(* Publish stable source identities and the complete typed Sequence status. *)
stMotionIntent.udiZCommandId := udiZCommandId;
stMotionIntent.udiRCommandId := udiRCommandId;
GVL_Status.stFast.stSequence.nAcceptedCommandId := udiActiveStartCommandId;
GVL_Status.stFast.stSequence.bBusy := bBusy;
GVL_Status.stFast.stSequence.bDone := bDone;
GVL_Status.stFast.stSequence.bAborted := bAborted;
GVL_Status.stFast.stSequence.bError := bError;
GVL_Status.stFast.stSequence.nErrorId := udiFirstFaultId;
GVL_Status.stFast.stSequence.eState := eNextState;
GVL_Status.stFast.stSequence.eStep := eStep;
GVL_Status.stFast.stSequence.eSubPhase := eSubPhase;
GVL_Status.stFast.stSequence.eEndCause := eEndCause;
GVL_Status.stFast.stSequence.eExitIntent := eExitIntent;
GVL_Status.stFast.stSequence.bCycleNok := bCycleNokLatched;
GVL_Status.stFast.stSequence.bRpmStopped := bRpmStopped;
GVL_Status.stFast.stSequence.bForceInBand := bForceInBand;
GVL_Status.stFast.stSequence.rStepTime_s := rStepTime_s;
GVL_Status.stFast.stSequence.rQualifiedForceHoldTime_s := rQualifiedForceHoldTime_s;
GVL_Status.stFast.stSequence.rForceSet_kN := rForceSet_kN;
GVL_Status.stFast.stSequence.rForceRamp_kN_s := rForceRamp_kN_s;
GVL_Status.stFast.stSequence.bForceControlEnable := bForceControlEnable;
GVL_Status.stFast.stSequence.bForceProfileTransfer := bForceProfileTransfer;
GVL_Status.stFast.stSequence.rForceTransferVelocity_mm_s := rForceTransferVelocity_mm_s;
GVL_Status.stFast.stSequence.rTargetRelativePosition_mm := rTargetRelativePosition_mm;
GVL_Status.stFast.stSequence.rHardMaximumRelativePosition_mm := rHardMaximumRelativePosition_mm;
GVL_Status.stFast.stSequence.bForceHardLimitActive := bHardForceActive;
GVL_Status.stFast.stSequence.bStrokeHardLimitActive := bHardStrokeActive;
GVL_Status.stFast.stSequence.bCollisionLimitActive := bCollisionLimitActive;
GVL_Status.stFast.stSequence.rSpeedSet_rpm := rSpeedSet_rpm;
GVL_Status.stFast.stSequence.stContact := fbContactDetect.stOutput;
GVL_Status.stFast.stSequence.stForceDecline := fbForceDecline.stOutput;
GVL_Status.stFast.stSequence.stStepCriterion := fbStepCriterion.stOutput;
GVL_Status.stFast.stSequence.stMotionIntent := stMotionIntent;
GVL_Status.stFast.stSequence.stFastConfigSnapshot := stFastConfigSnapshot;

GVL_Alarm.astRequests[9].eCode := E_AlarmCode.ALARM_CFF_CRITERION_FAULT;
GVL_Alarm.astRequests[9].eLevel := E_AlarmLevel.ALARM_LEVEL_FAULT;
GVL_Alarm.astRequests[9].nTextId := 3000;
GVL_Alarm.astRequests[9].nSourceId := 9;
GVL_Alarm.astRequests[9].bLatch := TRUE;
GVL_Alarm.astRequests[9].bActive := fbContactDetect.stOutput.bFault
    OR fbForceDecline.stOutput.bFault
    OR fbStepCriterion.stOutput.bFault;
GVL_Alarm.astRequests[10].eCode := E_AlarmCode.ALARM_CFF_SEQUENCE_FAULT;
GVL_Alarm.astRequests[10].eLevel := E_AlarmLevel.ALARM_LEVEL_FAULT;
GVL_Alarm.astRequests[10].nTextId := 3200;
GVL_Alarm.astRequests[10].nSourceId := 10;
GVL_Alarm.astRequests[10].bLatch := TRUE;
GVL_Alarm.astRequests[10].bActive := udiFirstFaultId <> 0;

(* Exactly one state assignment completes the scan. *)
ePreviousState := eState;
eState := eNextState;
bStateEntry := eState <> ePreviousState;

END_PROGRAM

// ---- POUs/FunctionBlocks/Control/FB_ForceDeclineObserver.TcPOU
FUNCTION_BLOCK FB_ForceDeclineObserver
VAR_INPUT
    (* 调用者完整赋值的Force Decline输入。 *)
    stInput : ST_ForceDeclineInput;
END_VAR
VAR_OUTPUT
    (* Arm、候选、确认、导数、锁存和故障输出。 *)
    stOutput : ST_ForceDeclineOutput;
END_VAR
VAR
    (* 当前步骤已经达到Arm Force。 *)
    bArmed : BOOL;
    (* 当前保持Decline回差候选。 *)
    bCandidate : BOOL;
    (* Decline已经连续确认。 *)
    bConfirmed : BOOL;
    (* 已获得上一个有效力样本。 *)
    bPreviousSampleValid : BOOL;
    (* 当前扫描满足全部Decline确认条件。 *)
    bDeclineCondition : BOOL;
    (* 当前配置和输入均有效。 *)
    bConfigurationValid : BOOL;
    (* 算法故障锁存；只有显式Reset清除。 *)
    bFaultLatched : BOOL;
    (* 已锁存的确定性故障编号。 *)
    udiLatchedFaultId : UDINT;
    (* 上一个有效力样本，单位kN。 *)
    rPreviousForce_kN : LREAL;
    (* 相邻样本力变化率，单位kN/s。 *)
    rForceDerivative_kN_s : LREAL;
    (* 连续确认累计时间，单位s。 *)
    rStableTime_s : LREAL;
    (* 确认锁存力，单位kN。 *)
    rLatchedForce_kN : LREAL;
    (* 确认锁存累计S_rel，单位mm。 *)
    rLatchedRelativePosition_mm : LREAL;
    (* 确认锁存主轴转速，单位rpm。 *)
    rLatchedSpeed_rpm : LREAL;
    (* 确认锁存步骤时间，单位s。 *)
    rLatchedStepTime_s : LREAL;
END_VAR

(* ---------------------------------------------------------
   Force Decline观察器。
   进入：步骤选择Decline主判据并提供有效ForceCriterion、RPM、S_rel和速度。
   动作：先Arm，再要求负下降率、窗口、捕获速度和连续Debounce。
   成功：锁存确认事实；不关闭PI、不切换Profile、不写流程状态。
   Fault：配置、信号或数值无效时锁存，只有显式Reset清除。
   --------------------------------------------------------- *)
IF stInput.bReset THEN
    bArmed := FALSE;
    bCandidate := FALSE;
    bConfirmed := FALSE;
    bPreviousSampleValid := FALSE;
    bFaultLatched := FALSE;
    udiLatchedFaultId := 0;
    rPreviousForce_kN := 0.0;
    rForceDerivative_kN_s := 0.0;
    rStableTime_s := 0.0;
    rLatchedForce_kN := 0.0;
    rLatchedRelativePosition_mm := 0.0;
    rLatchedSpeed_rpm := 0.0;
    rLatchedStepTime_s := 0.0;
ELSIF NOT stInput.bEnable THEN
    (* Disable结束当前步骤观察窗口，但故障保持到Reset。 *)
    bArmed := FALSE;
    bCandidate := FALSE;
    bConfirmed := FALSE;
    bPreviousSampleValid := FALSE;
    rForceDerivative_kN_s := 0.0;
    rStableTime_s := 0.0;
ELSIF NOT bFaultLatched AND NOT bConfirmed THEN
    bConfigurationValid := stInput.bSignalValid
        AND FC_IsFiniteLReal(rValue := stInput.rForceActual_kN)
        AND FC_IsFiniteLReal(rValue := stInput.rSpeed_rpm)
        AND FC_IsFiniteLReal(rValue := stInput.rRelativePosition_mm)
        AND FC_IsFiniteLReal(rValue := stInput.rAxisVelocity_mm_s)
        AND FC_IsFiniteLReal(rValue := stInput.rStepTime_s)
        AND FC_IsFiniteLReal(rValue := stInput.rArmForce_kN)
        AND FC_IsFiniteLReal(rValue := stInput.rDeclineTo_kN)
        AND FC_IsFiniteLReal(rValue := stInput.rHysteresis_kN)
        AND FC_IsFiniteLReal(rValue := stInput.rMinimumDeclineRate_kN_s)
        AND FC_IsFiniteLReal(rValue := stInput.rCriterionSRelMinimum_mm)
        AND FC_IsFiniteLReal(rValue := stInput.rCriterionSRelMaximum_mm)
        AND FC_IsFiniteLReal(rValue := stInput.rCriterionRpmMinimum)
        AND FC_IsFiniteLReal(rValue := stInput.rCaptureMaximumVelocity_mm_s)
        AND FC_IsFiniteLReal(rValue := stInput.rDebounceTime_s)
        AND FC_IsFiniteLReal(rValue := stInput.rCycleTime_s)
        AND (stInput.rDeclineTo_kN >= 0.0)
        AND (stInput.rHysteresis_kN >= 0.0)
        AND (stInput.rArmForce_kN > stInput.rDeclineTo_kN + stInput.rHysteresis_kN)
        AND (stInput.rMinimumDeclineRate_kN_s > 0.0)
        AND (stInput.rCriterionSRelMaximum_mm >= stInput.rCriterionSRelMinimum_mm)
        AND (stInput.rCriterionRpmMinimum >= 0.0)
        AND (stInput.rCaptureMaximumVelocity_mm_s > 0.0)
        AND (stInput.rDebounceTime_s > 0.0)
        AND (stInput.rCycleTime_s > 0.0);

    IF NOT bConfigurationValid THEN
        bFaultLatched := TRUE;
        udiLatchedFaultId := 16#00009101;
    ELSE
        IF bPreviousSampleValid THEN
            rForceDerivative_kN_s := (stInput.rForceActual_kN - rPreviousForce_kN)
                / stInput.rCycleTime_s;
            IF NOT FC_IsFiniteLReal(rValue := rForceDerivative_kN_s) THEN
                bFaultLatched := TRUE;
                udiLatchedFaultId := 16#00009102;
            END_IF
        ELSE
            rForceDerivative_kN_s := 0.0;
            bPreviousSampleValid := TRUE;
        END_IF
        rPreviousForce_kN := stInput.rForceActual_kN;

        IF NOT bFaultLatched THEN
            IF stInput.rForceActual_kN >= stInput.rArmForce_kN THEN
                bArmed := TRUE;
            END_IF

            IF NOT bCandidate AND bArmed
                AND (stInput.rForceActual_kN <= stInput.rDeclineTo_kN) THEN
                bCandidate := TRUE;
            END_IF

            IF bCandidate AND (stInput.rForceActual_kN
                > stInput.rDeclineTo_kN + stInput.rHysteresis_kN) THEN
                bCandidate := FALSE;
                rStableTime_s := 0.0;
            ELSE
                bDeclineCondition := bCandidate
                    AND (stInput.rForceActual_kN <= stInput.rDeclineTo_kN)
                    AND (rForceDerivative_kN_s <= -ABS(stInput.rMinimumDeclineRate_kN_s))
                    AND (stInput.rRelativePosition_mm >= stInput.rCriterionSRelMinimum_mm)
                    AND (stInput.rRelativePosition_mm <= stInput.rCriterionSRelMaximum_mm)
                    AND (ABS(stInput.rSpeed_rpm) >= ABS(stInput.rCriterionRpmMinimum))
                    AND (ABS(stInput.rAxisVelocity_mm_s) <= ABS(stInput.rCaptureMaximumVelocity_mm_s));

                IF bDeclineCondition THEN
                    rStableTime_s := rStableTime_s + stInput.rCycleTime_s;
                    IF NOT FC_IsFiniteLReal(rValue := rStableTime_s) THEN
                        bFaultLatched := TRUE;
                        udiLatchedFaultId := 16#00009103;
                    ELSIF rStableTime_s >= stInput.rDebounceTime_s THEN
                        bCandidate := FALSE;
                        bConfirmed := TRUE;
                        rLatchedForce_kN := stInput.rForceActual_kN;
                        rLatchedRelativePosition_mm := stInput.rRelativePosition_mm;
                        rLatchedSpeed_rpm := stInput.rSpeed_rpm;
                        rLatchedStepTime_s := stInput.rStepTime_s;
                    END_IF
                ELSE
                    (* 任一连续确认条件中断均清零Debounce；候选只由Force回差释放。 *)
                    rStableTime_s := 0.0;
                END_IF
            END_IF
        END_IF
    END_IF
END_IF

stOutput.bArmed := bArmed;
stOutput.bCandidate := bCandidate;
stOutput.bConfirmed := bConfirmed;
stOutput.rForceDerivative_kN_s := rForceDerivative_kN_s;
stOutput.rStableTime_s := rStableTime_s;
stOutput.rLatchedForce_kN := rLatchedForce_kN;
stOutput.rLatchedRelativePosition_mm := rLatchedRelativePosition_mm;
stOutput.rLatchedSpeed_rpm := rLatchedSpeed_rpm;
stOutput.rLatchedStepTime_s := rLatchedStepTime_s;
stOutput.bFault := bFaultLatched;
stOutput.nFaultId := udiLatchedFaultId;

END_FUNCTION_BLOCK

// ---- POUs/FunctionBlocks/Control/FB_StepProceedingCriterion.TcPOU
FUNCTION_BLOCK FB_StepProceedingCriterion
VAR_INPUT
    (* 调用者完整赋值的步骤推进输入。 *)
    stInput : ST_StepCriterionInput;
END_VAR
VAR_OUTPUT
    (* 步骤结束事实、动作、锁存和故障输出。 *)
    stOutput : ST_StepCriterionOutput;
END_VAR
VAR
    (* 当前Primary已经满足。 *)
    bPrimaryMet : BOOL;
    (* 当前Primary需要累计S_rel Secondary。 *)
    bSecondaryRequired : BOOL;
    (* 本扫描输入数值和配置有效。 *)
    bConfigurationValid : BOOL;
    (* 算法故障锁存；只有显式Reset清除。 *)
    bFaultLatched : BOOL;
    (* 已锁存的确定性故障编号。 *)
    udiLatchedFaultId : UDINT;
END_VAR

(* ---------------------------------------------------------
   步骤推进判据。
   进入：单一Primary、可选累计S_rel Secondary、StepMin/Max和硬原因有效。
   动作：安全原因和Secondary优先，Primary满足立即结束，StepMax只监视未满足Primary。
   成功：锁存EndCause、Force、S_rel、时间和流程动作。
   Fault：配置、数值或未知枚举无效时锁存，只有显式Reset清除。
   --------------------------------------------------------- *)
IF stInput.bReset THEN
    stOutput.bArmed := FALSE;
    stOutput.bPrimaryMet := FALSE;
    stOutput.bSecondaryLimitReached := FALSE;
    stOutput.bEndConfirmed := FALSE;
    stOutput.bTooShort := FALSE;
    stOutput.bNok := FALSE;
    stOutput.bAdvanceRequested := FALSE;
    stOutput.bControlledExitRequested := FALSE;
    stOutput.bDownwardMotionInhibited := FALSE;
    stOutput.eEndCause := STEP_END_NONE;
    stOutput.rLatchedForce_kN := 0.0;
    stOutput.rLatchedRelativePosition_mm := 0.0;
    stOutput.rLatchedStepTime_s := 0.0;
    stOutput.bFault := FALSE;
    stOutput.nFaultId := 0;
    bFaultLatched := FALSE;
    udiLatchedFaultId := 0;
    RETURN;
END_IF

IF NOT stInput.bEnable THEN
    stOutput.bArmed := FALSE;
    RETURN;
END_IF

stOutput.bArmed := stInput.bForceDeclineArmed;
IF bFaultLatched THEN
    stOutput.bEndConfirmed := TRUE;
    stOutput.bNok := TRUE;
    stOutput.bAdvanceRequested := FALSE;
    stOutput.bControlledExitRequested := TRUE;
    stOutput.bDownwardMotionInhibited := TRUE;
    stOutput.eEndCause := STEP_END_NONE;
    stOutput.bFault := TRUE;
    stOutput.nFaultId := udiLatchedFaultId;
    RETURN;
END_IF
IF stOutput.bEndConfirmed THEN
    RETURN;
END_IF

bConfigurationValid := FC_IsFiniteLReal(rValue := stInput.rRelativePosition_mm)
    AND FC_IsFiniteLReal(rValue := stInput.rRelativeDistanceTarget_mm)
    AND FC_IsFiniteLReal(rValue := stInput.rStepTime_s)
    AND FC_IsFiniteLReal(rValue := stInput.rStepTimeTarget_s)
    AND FC_IsFiniteLReal(rValue := stInput.rStepMinimumTime_s)
    AND FC_IsFiniteLReal(rValue := stInput.rStepMaximumTime_s)
    AND FC_IsFiniteLReal(rValue := stInput.rForceActual_kN)
    AND FC_IsFiniteLReal(rValue := stInput.rSecondaryDistanceLimit_mm)
    AND (stInput.rStepTime_s >= 0.0)
    AND (stInput.rStepMinimumTime_s >= 0.0)
    AND (stInput.rStepMaximumTime_s > 0.0)
    AND (stInput.rStepMinimumTime_s <= stInput.rStepMaximumTime_s)
    AND NOT (stInput.bForceDeclineConfirmed AND NOT stInput.bForceDeclineArmed);
IF NOT bConfigurationValid THEN
    bFaultLatched := TRUE;
    udiLatchedFaultId := 16#00009201;
END_IF
IF bFaultLatched THEN
    stOutput.bEndConfirmed := TRUE;
    stOutput.bNok := TRUE;
    stOutput.bAdvanceRequested := FALSE;
    stOutput.bControlledExitRequested := TRUE;
    stOutput.bDownwardMotionInhibited := TRUE;
    stOutput.eEndCause := STEP_END_NONE;
    stOutput.bFault := TRUE;
    stOutput.nFaultId := udiLatchedFaultId;
    RETURN;
END_IF

CASE stInput.ePrimaryCriterion OF
    STEP_CRIT_RELATIVE_DISTANCE:
        bSecondaryRequired := FALSE;
        bPrimaryMet := stInput.rRelativePosition_mm >= stInput.rRelativeDistanceTarget_mm;
        IF stInput.rRelativeDistanceTarget_mm <= 0.0 THEN
            bFaultLatched := TRUE;
            udiLatchedFaultId := 16#00009202;
        END_IF
    STEP_CRIT_STEP_TIME:
        bSecondaryRequired := TRUE;
        bPrimaryMet := stInput.rStepTime_s >= stInput.rStepTimeTarget_s;
        IF (stInput.rStepTimeTarget_s <= 0.0)
            OR (stInput.rStepTimeTarget_s < stInput.rStepMinimumTime_s)
            OR (stInput.rStepTimeTarget_s > stInput.rStepMaximumTime_s)
            OR (stInput.rSecondaryDistanceLimit_mm <= 0.0) THEN
            bFaultLatched := TRUE;
            udiLatchedFaultId := 16#00009203;
        END_IF
    STEP_CRIT_FORCE_DECLINE_TO:
        bSecondaryRequired := TRUE;
        bPrimaryMet := stInput.bForceDeclineConfirmed;
        IF stInput.rSecondaryDistanceLimit_mm <= 0.0 THEN
            bFaultLatched := TRUE;
            udiLatchedFaultId := 16#00009204;
        END_IF
ELSE
    bFaultLatched := TRUE;
    udiLatchedFaultId := 16#00009205;
END_CASE

IF NOT bFaultLatched AND bSecondaryRequired THEN
    CASE stInput.eSecondaryAction OF
        SECONDARY_ADVANCE_AND_NOK:
        SECONDARY_CONTROLLED_EXIT_NOK:
    ELSE
        bFaultLatched := TRUE;
        udiLatchedFaultId := 16#00009206;
    END_CASE
END_IF
IF bFaultLatched THEN
    stOutput.bEndConfirmed := TRUE;
    stOutput.bNok := TRUE;
    stOutput.bAdvanceRequested := FALSE;
    stOutput.bControlledExitRequested := TRUE;
    stOutput.bDownwardMotionInhibited := TRUE;
    stOutput.eEndCause := STEP_END_NONE;
    stOutput.bFault := TRUE;
    stOutput.nFaultId := udiLatchedFaultId;
    RETURN;
END_IF

(* EVAL_STAGE_HARD_CAUSE：Stop、轴、传感器和硬边界拥有最高优先级。 *)
IF stInput.bStopRequested THEN
    stOutput.bEndConfirmed := TRUE;
    stOutput.bNok := TRUE;
    stOutput.bControlledExitRequested := TRUE;
    stOutput.bDownwardMotionInhibited := TRUE;
    stOutput.eEndCause := STEP_END_STOP_REQUEST;
ELSIF stInput.bAxisFault THEN
    stOutput.bEndConfirmed := TRUE;
    stOutput.bNok := TRUE;
    stOutput.bControlledExitRequested := TRUE;
    stOutput.bDownwardMotionInhibited := TRUE;
    stOutput.eEndCause := STEP_END_AXIS_FAULT;
ELSIF stInput.bSensorInvalid OR NOT stInput.bSignalValid THEN
    stOutput.bEndConfirmed := TRUE;
    stOutput.bNok := TRUE;
    stOutput.bControlledExitRequested := TRUE;
    stOutput.bDownwardMotionInhibited := TRUE;
    stOutput.eEndCause := STEP_END_SENSOR_INVALID;
ELSIF stInput.bCollisionActive THEN
    stOutput.bEndConfirmed := TRUE;
    stOutput.bNok := TRUE;
    stOutput.bControlledExitRequested := TRUE;
    stOutput.bDownwardMotionInhibited := TRUE;
    stOutput.eEndCause := STEP_END_COLLISION;
ELSIF stInput.bHardForceActive THEN
    stOutput.bEndConfirmed := TRUE;
    stOutput.bNok := TRUE;
    stOutput.bControlledExitRequested := TRUE;
    stOutput.bDownwardMotionInhibited := TRUE;
    stOutput.eEndCause := STEP_END_HARD_FORCE;
ELSIF stInput.bHardStrokeActive THEN
    stOutput.bEndConfirmed := TRUE;
    stOutput.bNok := TRUE;
    stOutput.bControlledExitRequested := TRUE;
    stOutput.bDownwardMotionInhibited := TRUE;
    stOutput.eEndCause := STEP_END_HARD_STROKE;
END_IF

(* EVAL_STAGE_SECONDARY：累计S_rel先于Primary处理并立即禁止继续向下。 *)
IF NOT stOutput.bEndConfirmed AND bSecondaryRequired
    AND (stInput.rRelativePosition_mm >= stInput.rSecondaryDistanceLimit_mm) THEN
    stOutput.bSecondaryLimitReached := TRUE;
    stOutput.bEndConfirmed := TRUE;
    stOutput.bNok := TRUE;
    stOutput.bDownwardMotionInhibited := TRUE;
    stOutput.eEndCause := STEP_END_SECONDARY_RELATIVE_DISTANCE;
    CASE stInput.eSecondaryAction OF
        SECONDARY_ADVANCE_AND_NOK:
            stOutput.bAdvanceRequested := TRUE;
        SECONDARY_CONTROLLED_EXIT_NOK:
            stOutput.bControlledExitRequested := TRUE;
    END_CASE
END_IF

(* EVAL_STAGE_PRIMARY：Primary一旦满足立即结束，StepMin只判质量。 *)
IF NOT stOutput.bEndConfirmed AND bPrimaryMet THEN
    stOutput.bPrimaryMet := TRUE;
    stOutput.bEndConfirmed := TRUE;
    stOutput.bAdvanceRequested := TRUE;
    stOutput.eEndCause := FC_GetPrimaryEndCause(ePrimaryCriterion := stInput.ePrimaryCriterion);
    IF stInput.rStepTime_s < stInput.rStepMinimumTime_s THEN
        stOutput.bTooShort := TRUE;
        stOutput.bNok := TRUE;
    END_IF
END_IF

(* EVAL_STAGE_STEP_MAX：仅在Primary未满足时触发等待看门狗。 *)
IF NOT stOutput.bEndConfirmed AND (stInput.rStepTime_s >= stInput.rStepMaximumTime_s) THEN
    stOutput.bEndConfirmed := TRUE;
    stOutput.bNok := TRUE;
    stOutput.bControlledExitRequested := TRUE;
    stOutput.bDownwardMotionInhibited := TRUE;
    stOutput.eEndCause := STEP_END_MAX_TIME;
END_IF

IF stOutput.bEndConfirmed THEN
    stOutput.rLatchedForce_kN := stInput.rForceActual_kN;
    stOutput.rLatchedRelativePosition_mm := stInput.rRelativePosition_mm;
    stOutput.rLatchedStepTime_s := stInput.rStepTime_s;
END_IF
stOutput.bFault := bFaultLatched;
stOutput.nFaultId := udiLatchedFaultId;

END_FUNCTION_BLOCK

// ---- POUs/Functions/FC_ValidateJoinProgram.TcPOU
FUNCTION FC_ValidateJoinProgram : BOOL
VAR_INPUT
    (* 待校验的四步骤连接程序。 *)
    stProgram : ST_CffJoinProgram;
    (* 机器硬限制；程序值不得超过这些边界。 *)
    stMachineLimits : ST_MachineLimits;
END_VAR
VAR
    (* 固定四步骤遍历索引。 *)
    nStepIndex : INT;
    (* 当前步骤的局部副本。 *)
    stStep : ST_CffStepProgram;
    (* 上一步骤允许到达的累计S_rel边界，单位mm。 *)
    rPreviousStepBoundary_mm : LREAL;
    (* 当前步骤Primary或Secondary对应的累计S_rel边界，单位mm。 *)
    rCurrentStepBoundary_mm : LREAL;
    (* Z轴绝对软限位跨度，作为累计S_rel程序上限，单位mm。 *)
    rMaximumRelativeTravel_mm : LREAL;
    (* 第四步的局部副本。*)
    stStep4 : ST_CffStepProgram;
    (* 第四步合格力带保持时间，单位毫秒。*)
    nQualifiedForceHoldMs : UDINT;
    (* 第四步主时间判据，单位毫秒。*)
    nPrimaryStepTimeMs : UDINT;
END_VAR

FC_ValidateJoinProgram := FALSE;
rPreviousStepBoundary_mm := 0.0;
rMaximumRelativeTravel_mm := ABS(stMachineLimits.fZMaxPositionMm
    - stMachineLimits.fZMinPositionMm);

(* 程序、机器限值、Contact参数和受控修订必须先有效。 *)
IF NOT stProgram.bValid OR NOT stMachineLimits.bValid OR NOT stProgram.stMonitor.bValid
    OR (stProgram.stHeader.nProgramId = 0)
    OR (stProgram.stHeader.nRevision = 0)
    OR (stProgram.stHeader.nElementTypeId = 0)
    OR NOT (stProgram.stHeader.nForceProfileId > 0)
    OR NOT (stProgram.stHeader.nRAxisProfileId > 0)
    OR (stProgram.stHeader.nToolId = 0)
    OR (stProgram.stHeader.nAnvilId = 0)
    OR (stMachineLimits.fMaxForceN <= 0.0)
    OR (stMachineLimits.fRMaxSpeedRpm <= 0.0)
    OR (stMachineLimits.fZMaxVelocityMmS <= 0.0)
    OR (stMachineLimits.fZMaxPositionMm <= stMachineLimits.fZMinPositionMm)
    OR NOT FC_IsFiniteLReal(rValue := stMachineLimits.fMaxForceN)
    OR NOT FC_IsFiniteLReal(rValue := stMachineLimits.fRMaxSpeedRpm)
    OR NOT FC_IsFiniteLReal(rValue := stMachineLimits.fZMinPositionMm)
    OR NOT FC_IsFiniteLReal(rValue := stMachineLimits.fZMaxPositionMm)
    OR NOT FC_IsFiniteLReal(rValue := stMachineLimits.fZMaxVelocityMmS)
    OR NOT FC_IsFiniteLReal(rValue := rMaximumRelativeTravel_mm)
    OR NOT FC_IsFiniteLReal(rValue := stProgram.stHeader.fMaterialThicknessMm)
    OR NOT FC_IsFiniteLReal(rValue := stProgram.stHeader.fThicknessToleranceMm)
    OR NOT FC_IsFiniteLReal(rValue := stProgram.stHeader.fContactForceOnN)
    OR NOT FC_IsFiniteLReal(rValue := stProgram.stHeader.fContactForceOffN)
    OR NOT FC_IsFiniteLReal(rValue := stProgram.stHeader.fContactSearchVelocityMmS)
    OR NOT FC_IsFiniteLReal(rValue := stProgram.stHeader.fContactSearchStartPositionMm)
    OR NOT FC_IsFiniteLReal(rValue := stProgram.stHeader.fContactSensorMinimumMm)
    OR NOT FC_IsFiniteLReal(rValue := stProgram.stHeader.fContactSensorMaximumMm)
    OR NOT FC_IsFiniteLReal(rValue := stProgram.stHeader.fReturnVelocityMmS)
    OR NOT FC_IsFiniteLReal(rValue := stProgram.stHeader.fReturnOpeningMm)
    OR (stProgram.stHeader.fMaterialThicknessMm <= 0.0)
    OR (stProgram.stHeader.fThicknessToleranceMm < 0.0)
    OR (stProgram.stHeader.fContactForceOffN < 0.0)
    OR (stProgram.stHeader.fContactForceOnN <= stProgram.stHeader.fContactForceOffN)
    OR (stProgram.stHeader.fContactForceOnN >= stMachineLimits.fMaxForceN)
    OR (stProgram.stHeader.nContactDebounceMs = 0)
    OR (stProgram.stHeader.fContactSearchVelocityMmS <= 0.0)
    OR (stProgram.stHeader.fContactSearchVelocityMmS > stMachineLimits.fZMaxVelocityMmS)
    OR NOT (stProgram.stHeader.fContactSearchStartPositionMm >= stMachineLimits.fZMinPositionMm)
    OR NOT (stProgram.stHeader.fContactSearchStartPositionMm <= stMachineLimits.fZMaxPositionMm)
    OR (stProgram.stHeader.fContactSensorMaximumMm
        <= stProgram.stHeader.fContactSensorMinimumMm)
    OR (stProgram.stHeader.fReturnVelocityMmS <= 0.0)
    OR (stProgram.stHeader.fReturnVelocityMmS > stMachineLimits.fZMaxVelocityMmS)
    OR (stProgram.stHeader.fReturnOpeningMm < stMachineLimits.fZMinPositionMm)
    OR (stProgram.stHeader.fReturnOpeningMm > stMachineLimits.fZMaxPositionMm)
    OR ((stProgram.stHeader.eReturnMode <> RETURN_MODE_LOCAL)
        AND (stProgram.stHeader.eReturnMode <> RETURN_MODE_REFERENCE))
    OR ((stProgram.stHeader.eState <> PROGRAM_VALID)
        AND (stProgram.stHeader.eState <> PROGRAM_ACTIVE))
    OR NOT FC_IsFiniteLReal(rValue := stProgram.stMonitor.fMinForceN)
    OR NOT FC_IsFiniteLReal(rValue := stProgram.stMonitor.fMaxForceN)
    OR NOT FC_IsFiniteLReal(rValue := stProgram.stMonitor.fMinRelativeDistanceMm)
    OR NOT FC_IsFiniteLReal(rValue := stProgram.stMonitor.fMaxRelativeDistanceMm)
    OR NOT FC_IsFiniteLReal(rValue := stProgram.stMonitor.fMinTorqueNm)
    OR NOT FC_IsFiniteLReal(rValue := stProgram.stMonitor.fMaxTorqueNm)
    OR NOT FC_IsFiniteLReal(rValue := stProgram.stMonitor.fMinEnergyJ)
    OR NOT FC_IsFiniteLReal(rValue := stProgram.stMonitor.fMaxEnergyJ)
    OR (stProgram.stMonitor.fMinForceN > stProgram.stMonitor.fMaxForceN)
    OR (stProgram.stMonitor.fMaxForceN > stMachineLimits.fMaxForceN)
    OR (stProgram.stMonitor.fMinRelativeDistanceMm
        > stProgram.stMonitor.fMaxRelativeDistanceMm)
    OR (stProgram.stMonitor.fMinTorqueNm > stProgram.stMonitor.fMaxTorqueNm)
    OR (stProgram.stMonitor.fMinEnergyJ > stProgram.stMonitor.fMaxEnergyJ) THEN
    RETURN;
END_IF

FOR nStepIndex := 1 TO 4 DO
    stStep := stProgram.astSteps[nStepIndex];
    IF NOT stStep.bValid OR NOT stStep.stProceeding.bValid
        OR NOT FC_IsFiniteLReal(rValue := stStep.fSetForceN)
        OR NOT FC_IsFiniteLReal(rValue := stStep.fSetSpeedRpm)
        OR NOT FC_IsFiniteLReal(rValue := stStep.fForceRampNS)
        OR NOT FC_IsFiniteLReal(rValue := stStep.stProceeding.fRelativeDistanceMm)
        OR NOT FC_IsFiniteLReal(rValue := stStep.stProceeding.fSecondarySRelMm)
        OR NOT FC_IsFiniteLReal(rValue := stStep.stProceeding.fDeclineToN)
        OR NOT FC_IsFiniteLReal(rValue := stStep.stProceeding.fArmForceN)
        OR NOT FC_IsFiniteLReal(rValue := stStep.stProceeding.fDeclineHysteresisN)
        OR NOT FC_IsFiniteLReal(rValue := stStep.stProceeding.fMinimumDeclineRateNS)
        OR NOT FC_IsFiniteLReal(rValue := stStep.stProceeding.fCriterionSRelMinMm)
        OR NOT FC_IsFiniteLReal(rValue := stStep.stProceeding.fCriterionSRelMaxMm)
        OR NOT FC_IsFiniteLReal(rValue := stStep.stProceeding.fCriterionRpmMin)
        OR NOT FC_IsFiniteLReal(rValue := stStep.stProceeding.fCaptureMaxVelocityMmS)
        OR NOT FC_IsFiniteLReal(rValue := stStep.stProceeding.fForceBandToleranceN)
        OR NOT FC_IsFiniteLReal(rValue := stStep.stProceeding.fRpmStoppedThresholdRpm)
        OR (stStep.fSetForceN < 0.0)
        OR (stStep.fSetForceN >= stMachineLimits.fMaxForceN)
        OR (ABS(stStep.fSetSpeedRpm) > stMachineLimits.fRMaxSpeedRpm)
        OR (stStep.fForceRampNS <= 0.0)
        OR (stStep.nMonitorProfileId = 0)
        OR (stStep.stProceeding.nStepMaxMs = 0)
        OR (stStep.stProceeding.nStepMinMs > stStep.stProceeding.nStepMaxMs) THEN
        RETURN;
    END_IF

    (* 数组位置和显式步骤编号必须一致，防止配方步骤错位。 *)
    CASE nStepIndex OF
        1: IF stStep.eStep <> CFF_STEP1_PENETRATION THEN RETURN; END_IF
        2: IF stStep.eStep <> CFF_STEP2_CLEAN_ACTIVATE THEN RETURN; END_IF
        3: IF stStep.eStep <> CFF_STEP3_WELDING THEN RETURN; END_IF
        4: IF stStep.eStep <> CFF_STEP4_COMPRESSION THEN RETURN; END_IF
    END_CASE

    CASE stStep.stProceeding.ePrimaryCriterion OF
        STEP_CRIT_RELATIVE_DISTANCE:
            IF (stStep.stProceeding.fRelativeDistanceMm <= 0.0)
                OR (stStep.stProceeding.fSecondarySRelMm <> 0.0) THEN
                RETURN;
            END_IF
            rCurrentStepBoundary_mm := stStep.stProceeding.fRelativeDistanceMm;
        STEP_CRIT_STEP_TIME:
            IF (stStep.stProceeding.nPrimaryStepTimeMs = 0)
                OR (stStep.stProceeding.nPrimaryStepTimeMs < stStep.stProceeding.nStepMinMs)
                OR (stStep.stProceeding.nPrimaryStepTimeMs > stStep.stProceeding.nStepMaxMs)
                OR (stStep.stProceeding.fSecondarySRelMm <= 0.0) THEN
                RETURN;
            END_IF
            rCurrentStepBoundary_mm := stStep.stProceeding.fSecondarySRelMm;
        STEP_CRIT_FORCE_DECLINE_TO:
            IF (stStep.stProceeding.fDeclineToN < 0.0)
                OR (stStep.stProceeding.fDeclineToN >= stStep.fSetForceN)
                OR (stStep.stProceeding.fDeclineHysteresisN < 0.0)
                OR (stStep.stProceeding.fArmForceN
                    <= stStep.stProceeding.fDeclineToN
                        + stStep.stProceeding.fDeclineHysteresisN)
                OR (stStep.stProceeding.fArmForceN > stStep.fSetForceN)
                OR (stStep.stProceeding.fMinimumDeclineRateNS <= 0.0)
                OR (stStep.stProceeding.nDeclineDebounceMs = 0)
                OR (stStep.stProceeding.fCriterionSRelMinMm < 0.0)
                OR (stStep.stProceeding.fCriterionSRelMaxMm
                    < stStep.stProceeding.fCriterionSRelMinMm)
                OR (stStep.stProceeding.fSecondarySRelMm <= 0.0)
                OR (stStep.stProceeding.fCriterionSRelMaxMm
                    > stStep.stProceeding.fSecondarySRelMm)
                OR (stStep.stProceeding.fCriterionRpmMin < 0.0)
                OR (stStep.stProceeding.fCriterionRpmMin
                    > stMachineLimits.fRMaxSpeedRpm)
                OR (stStep.stProceeding.fCaptureMaxVelocityMmS <= 0.0)
                OR (stStep.stProceeding.fCaptureMaxVelocityMmS
                    > stMachineLimits.fZMaxVelocityMmS) THEN
                RETURN;
            END_IF
            rCurrentStepBoundary_mm := stStep.stProceeding.fSecondarySRelMm;
    ELSE
        RETURN;
    END_CASE

    CASE stStep.stProceeding.eSecondaryAction OF
        SECONDARY_ADVANCE_AND_NOK:
        SECONDARY_CONTROLLED_EXIT_NOK:
    ELSE
        RETURN;
    END_CASE

    (* 四步骤共用Contact零点，允许到达的累计S_rel不得回退或超过机器跨度。 *)
    IF (rCurrentStepBoundary_mm < rPreviousStepBoundary_mm)
        OR (rCurrentStepBoundary_mm > rMaximumRelativeTravel_mm) THEN
        RETURN;
    END_IF
    rPreviousStepBoundary_mm := rCurrentStepBoundary_mm;
END_FOR

(* 第四步只能以时间推进，并在压实前完成受控的合格力带保持。*)
stStep4 := stProgram.astSteps[4];
nQualifiedForceHoldMs := stStep4.stProceeding.nQualifiedForceHoldMs;
nPrimaryStepTimeMs := stStep4.stProceeding.nPrimaryStepTimeMs;
IF NOT (stStep4.stProceeding.ePrimaryCriterion = STEP_CRIT_STEP_TIME)
    OR NOT (nQualifiedForceHoldMs > 0)
    OR NOT (nQualifiedForceHoldMs <= nPrimaryStepTimeMs)
    OR NOT (stStep4.stProceeding.fForceBandToleranceN > 0.0)
    OR NOT (stStep4.stProceeding.fForceBandToleranceN < stMachineLimits.fMaxForceN)
    OR NOT (stStep4.stProceeding.fRpmStoppedThresholdRpm >= 0.0)
    OR NOT (stStep4.stProceeding.fRpmStoppedThresholdRpm < stMachineLimits.fRMaxSpeedRpm)
    OR NOT (stStep4.stProceeding.eSecondaryAction = SECONDARY_CONTROLLED_EXIT_NOK)
    OR NOT (stStep4.fSetSpeedRpm = 0.0) THEN
    RETURN;
END_IF

FC_ValidateJoinProgram := TRUE;

END_FUNCTION

// ---- POUs/Fast/PRG_FastAxisControl.TcPOU
PROGRAM PRG_FastAxisControl
VAR
    (* ---------------------------------------------------------
       Z轴命令Owner仲裁实例；活动Force Owner仅在Sequence意图和
       External Adapter均确认释放后才能转交。
       --------------------------------------------------------- *)
    fbZAxisArbiter : FB_AxisCommandArbiter;
    (* Force设定值、Profile无扰切换和导纳控制唯一实例。 *)
    fbForceSetpointRamp : FB_SetpointRamp;
    fbZProfileSwitch : FB_BumplessProfileSwitch;
    fbZForceAdmittance : FB_ZForceAdmittance;
    (* ---------------------------------------------------------
       Z轴External轨迹唯一实例。
       生命周期：只消费Adapter accepted包和当前Sequence冻结快照；
       Reset：只允许External释放、Z/R实际静止后的安全终态Reset。
       --------------------------------------------------------- *)
    fbZExternalTrajectory : FB_ZExternalTrajectory;
    (* ---------------------------------------------------------
       R轴软件速度包络唯一实例。
       生命周期：每个新Adapter事务从实际RPM初始化一次；稳定扫描只
       发布诊断包络，不把包络逐扫描转换成新的MC事务。
       --------------------------------------------------------- *)
    fbRSpeedRamp : FB_SetpointRamp;
    (* 唯一标准NC及External API Adapter实例。 *)
    fbZAxisNc : FB_ZAxisNcAdapter;
    fbZAxisExtSetpointAdapter : FB_ZAxisExtSetpointAdapter;
    fbRAxisNc : FB_RAxisNcAdapter;

    stHomeCommand : ST_ZAxisCommand;
    stManualCommand : ST_ZAxisCommand;
    stApproachCommand : ST_ZAxisCommand;
    stForceProcessCommand : ST_ZAxisCommand;
    stRetractCommand : ST_ZAxisCommand;
    stCandidateZSourceCommand : ST_ZAxisCommand;
    stLatchedZSourceCommand : ST_ZAxisCommand;
    stFaultStopCommand : ST_ZAxisCommand;
    stSelectedZCommand : ST_ZAxisCommand;
    stCandidateRSourceCommand : ST_RAxisCommand;
    stLatchedRAdapterCommand : ST_RAxisCommand;
    stSelectedRCommand : ST_RAxisCommand;
    stExtCommand : ST_ZExtSetpointCommand;
    stTrajectoryInput : ST_ZExternalTrajectoryInput;
    stZForceInput : ST_ZForceControlInput;

    bExternalCommandChannelBusy : BOOL;
    udiZStandardCommandId : UDINT;
    bFastConfigSnapshotCurrent : BOOL;
    bFastConfigSnapshotSeen : BOOL;
    bSequenceMotionIntentPresent : BOOL;
    bSnapshotMismatch : BOOL;
    bFastSafetyStopEvent : BOOL;
    bFastSafetyStopLatched : BOOL;
    bExternalSafelyReleasedForReset : BOOL;
    bSafeTerminalResetGatesMet : BOOL;
    bSafeTerminalReset : BOOL;
    bSafeTerminalResetRising : BOOL;
    bNewSafeTerminalSequenceCommand : BOOL;
    bNewSafeTerminalResetRequest : BOOL;
    bSafeTerminalResetPending : BOOL;
    bNormalZResetAllowed : BOOL;
    bLatchedZFaultStopRequest : BOOL;
    bForceProcessExitComplete : BOOL;
    bForceLoopRequested : BOOL;
    bForceInputsHealthy : BOOL;
    bForceRampInputValid : BOOL;
    bProfileTransferRequested : BOOL;
    bFastConfigSnapshotChanged : BOOL;
    bFastPathSafetyExit : BOOL;
    bHardOverrideRequested : BOOL;
    bHardOverrideStart : BOOL;
    bHardOverridePending : BOOL;
    bHardOverrideHandled : BOOL;
    bHardOverrideAccepted : BOOL;
    bHardOverridePackageExact : BOOL;
    rHardOverrideExpectedPosition_mm : LREAL;
    nHardOverrideExpectedDirection : DINT;
    udiHardOverrideAcceptedCounter : UDINT;

    bZSequenceSourceActive, bLastZSequenceSourceActive : BOOL;
    bRSequenceSourceActive, bLastRSequenceSourceActive : BOOL;
    udiLastZSourceCommandId, udiLastRSourceCommandId : UDINT;
    udiZAdapterCommandId, udiRAdapterCommandId : UDINT;
    udiCurrentSequenceZSourceId, udiCurrentSequenceRSourceId : UDINT;
    udiCurrentZSourceCommandId, udiCurrentRSourceCommandId : UDINT;
    udiAcceptedZSequenceSourceId, udiAcceptedRSequenceSourceId : UDINT;
    udiPendingZSequenceSourceId, udiPendingRSequenceSourceId : UDINT;
    udiPendingZAdapterCommandId, udiPendingRAdapterCommandId : UDINT;
    udiCurrentSafeTerminalResetRequestId : UDINT;
    udiLastObservedSafeTerminalSequenceCommandId : UDINT;
    udiPendingSafeTerminalResetRequestId : UDINT;
    udiConsumedSafeTerminalResetRequestId : UDINT;
    udiLastAppliedFastConfigCommandId : UDINT;
    bPendingZTransactionIsSequence, bPendingRTransactionIsSequence : BOOL;
    bNewZAdapterTransaction, bNewRAdapterTransaction : BOOL;
    bNewZSourceTransaction, bNewRSourceTransaction : BOOL;
    bPostResetZNormalBarrier, bPostResetRNormalBarrier : BOOL;
    bAcceptedFastPackageNewerThanReset : BOOL;
    bZNormalSourceBlockedByReset, bRNormalSourceBlockedByReset : BOOL;
    udiPostResetNormalBarrierRequestId : UDINT;
    bPendingRDecelerationValid : BOOL;
    bLastAcceptedRDecelerationValid : BOOL;
    rPendingRDeceleration_rpm_s : LREAL;
    rLastAcceptedRDeceleration_rpm_s : LREAL;
    bRSpeedRampSafeReset : BOOL;

    rForceActual_kN : LREAL;
    rFastCycleTime_s : LREAL;
    rEffectiveForceRamp_kN_s : LREAL;
    rForceRampRateForFb_kN_s : LREAL;
    rTrajectoryTargetVelocity_mm_s : LREAL;
END_VAR

(* Task_CffFast 中轴适配、External轨迹与力控仲裁的唯一Owner：PRG_FastAxisControl。 *)
(* ---------------------------------------------------------
   V3.7 Fast轴接线层。
   只消费FastInputs已接受命令和Sequence发布的一份冻结快照；
   算法FB不访问轴，所有MC调用仍由三个Adapter唯一拥有。
   --------------------------------------------------------- *)
bFastConfigSnapshotCurrent :=
    GVL_Status.stFast.stSequence.stFastConfigSnapshot.bValid
    AND GVL_Status.stFast.stSequence.stFastConfigSnapshot.nSequenceCommandId
        = GVL_Status.stFast.stSequence.nAcceptedCommandId;
bNewZAdapterTransaction := FALSE;
bNewRAdapterTransaction := FALSE;
rFastCycleTime_s := UDINT_TO_LREAL(
    GVL_Status.stFast.stSequence.stFastConfigSnapshot.stMachine.nFastTaskCycleUs)
    * 0.000001;

(* 安全终态Reset按accepted Sequence命令全事件高水位去重。
   命令可先锁存pending，待Release/Standstill门满足后只消费一次。 *)
bExternalSafelyReleasedForReset := fbZAxisExtSetpointAdapter.stStatus.bReleaseOwner
    OR (fbZAxisExtSetpointAdapter.stStatus.eState = E_ZExtSetpointState.Z_EXT_IDLE
        AND NOT fbZAxisExtSetpointAdapter.stStatus.bEnabled);
bSafeTerminalResetGatesMet := NOT GVL_Status.stFast.stSequence.bBusy
    AND bExternalSafelyReleasedForReset
    AND GVL_Status.stFast.stZAxis.bStandstill
    AND GVL_Status.stFast.stRAxis.bStandstill;
udiCurrentSafeTerminalResetRequestId :=
    GVL_FastInternal.stAcceptedCommand.stSequence.nCommandId;
bNewSafeTerminalSequenceCommand := FC_IsNewerRequestId(
    udiCandidate := udiCurrentSafeTerminalResetRequestId,
    udiReference := udiLastObservedSafeTerminalSequenceCommandId);
bNewSafeTerminalResetRequest := FALSE;
IF bNewSafeTerminalSequenceCommand THEN
    udiLastObservedSafeTerminalSequenceCommandId :=
        udiCurrentSafeTerminalResetRequestId;
    IF GVL_FastInternal.stAcceptedCommand.stSequence.bResetPulse THEN
        bNewSafeTerminalResetRequest := TRUE;
        udiPendingSafeTerminalResetRequestId :=
            udiCurrentSafeTerminalResetRequestId;
        bSafeTerminalResetPending := TRUE;
    END_IF
END_IF
bSafeTerminalReset := bSafeTerminalResetPending AND bSafeTerminalResetGatesMet;
bSafeTerminalResetRising := bSafeTerminalReset;
IF bSafeTerminalResetRising THEN
    bSafeTerminalResetPending := FALSE;
    udiConsumedSafeTerminalResetRequestId :=
        udiPendingSafeTerminalResetRequestId;
END_IF

(* 上一扫描R Adapter已接受且数值有效时，才更新Safety Stop减速度。 *)
IF bPendingRDecelerationValid
    AND (fbRAxisNc.udiAcceptedCommandId = udiPendingRAdapterCommandId)
    AND (udiPendingRAdapterCommandId <> 0) THEN
    rLastAcceptedRDeceleration_rpm_s := rPendingRDeceleration_rpm_s;
    bLastAcceptedRDecelerationValid := TRUE;
    bPendingRDecelerationValid := FALSE;
END_IF

(* PRECHECK允许Busy但尚未发布快照；只有见过快照或出现运动意图后失配才停机。 *)
IF bFastConfigSnapshotCurrent AND GVL_Status.stFast.stSequence.bBusy THEN
    bFastConfigSnapshotSeen := TRUE;
END_IF
IF bSafeTerminalResetRising THEN
    bFastConfigSnapshotSeen := FALSE;
END_IF
bSequenceMotionIntentPresent :=
    (GVL_Status.stFast.stSequence.stMotionIntent.stZCommand.eOwnerRequest
        <> E_ZCommandOwner.Z_OWNER_NONE)
    OR GVL_Status.stFast.stSequence.stMotionIntent.bRAxisProcessRequested
    OR GVL_Status.stFast.stSequence.stMotionIntent.bExternalEnableRequest
    OR GVL_Status.stFast.stSequence.stMotionIntent.bExternalDisableRequest
    OR GVL_Status.stFast.stSequence.bForceControlEnable;
bSnapshotMismatch := NOT bFastConfigSnapshotCurrent
    AND (bFastConfigSnapshotSeen OR bSequenceMotionIntentPresent);
bFastSafetyStopEvent := bSnapshotMismatch
    AND NOT bFastSafetyStopLatched
    AND NOT bSafeTerminalResetRising;
IF bFastSafetyStopEvent THEN
    bFastSafetyStopLatched := TRUE;
END_IF

(* 普通命令候选只从已接受命令区读取；Sequence按Owner精确覆盖。 *)
stCandidateZSourceCommand := GVL_FastInternal.stAcceptedCommand.stZAxis;
bZSequenceSourceActive := FALSE;
CASE GVL_Status.stFast.stSequence.stMotionIntent.stZCommand.eOwnerRequest OF
    E_ZCommandOwner.Z_OWNER_APPROACH:
        bZSequenceSourceActive := TRUE;
        stCandidateZSourceCommand :=
            GVL_Status.stFast.stSequence.stMotionIntent.stZCommand;
    E_ZCommandOwner.Z_OWNER_FORCE_PROCESS:
        bZSequenceSourceActive := TRUE;
        stCandidateZSourceCommand :=
            GVL_Status.stFast.stSequence.stMotionIntent.stZCommand;
    E_ZCommandOwner.Z_OWNER_RETRACT:
        bZSequenceSourceActive := TRUE;
        stCandidateZSourceCommand :=
            GVL_Status.stFast.stSequence.stMotionIntent.stZCommand;
    E_ZCommandOwner.Z_OWNER_FAULT_STOP:
        bZSequenceSourceActive := TRUE;
        stCandidateZSourceCommand :=
            GVL_Status.stFast.stSequence.stMotionIntent.stZCommand;
END_CASE
udiCurrentSequenceZSourceId :=
    GVL_Status.stFast.stSequence.stMotionIntent.udiZCommandId;
IF bZSequenceSourceActive THEN
    udiCurrentZSourceCommandId := udiCurrentSequenceZSourceId;
ELSE
    udiCurrentZSourceCommandId := GVL_FastInternal.stAcceptedCommand.nRequestId;
END_IF

(* Resolve the current R source before any central safety transaction. *)
bRSequenceSourceActive :=
    GVL_Status.stFast.stSequence.stMotionIntent.bRAxisProcessRequested;
udiCurrentSequenceRSourceId :=
    GVL_Status.stFast.stSequence.stMotionIntent.udiRCommandId;
IF bRSequenceSourceActive THEN
    stCandidateRSourceCommand :=
        GVL_Status.stFast.stSequence.stMotionIntent.stRCommand;
    udiCurrentRSourceCommandId := udiCurrentSequenceRSourceId;
ELSE
    stCandidateRSourceCommand := GVL_FastInternal.stAcceptedCommand.stRAxis;
    udiCurrentRSourceCommandId := GVL_FastInternal.stAcceptedCommand.nRequestId;
END_IF

bAcceptedFastPackageNewerThanReset := FC_IsNewerRequestId(
    udiCandidate := GVL_FastInternal.stAcceptedCommand.nRequestId,
    udiReference := udiPostResetNormalBarrierRequestId);
bZNormalSourceBlockedByReset := bPostResetZNormalBarrier
    AND NOT bAcceptedFastPackageNewerThanReset;
bNewZSourceTransaction := (udiCurrentZSourceCommandId <> 0)
    AND ((bZSequenceSourceActive <> bLastZSequenceSourceActive)
        OR FC_IsNewerRequestId(
            udiCandidate := udiCurrentZSourceCommandId,
            udiReference := udiLastZSourceCommandId));
IF bZNormalSourceBlockedByReset THEN
    bNewZSourceTransaction := FALSE;
END_IF
bNewZAdapterTransaction := FALSE;
IF NOT bFastSafetyStopLatched AND NOT bSafeTerminalResetRising THEN
    bNewZAdapterTransaction := bNewZSourceTransaction;
END_IF
IF bNewZAdapterTransaction THEN
    udiZAdapterCommandId := udiZAdapterCommandId + 1;
    IF udiZAdapterCommandId = 0 THEN
        udiZAdapterCommandId := 1;
    END_IF
    udiLastZSourceCommandId := udiCurrentZSourceCommandId;
    stLatchedZSourceCommand := stCandidateZSourceCommand;
    bLastZSequenceSourceActive := bZSequenceSourceActive;
    udiPendingZAdapterCommandId := udiZAdapterCommandId;
    bPendingZTransactionIsSequence := bZSequenceSourceActive;
    IF bZSequenceSourceActive THEN
        udiPendingZSequenceSourceId := udiCurrentSequenceZSourceId;
    ELSE
        udiPendingZSequenceSourceId := 0;
    END_IF
    IF bPostResetZNormalBarrier
        AND NOT bZSequenceSourceActive
        AND bAcceptedFastPackageNewerThanReset THEN
        bPostResetZNormalBarrier := FALSE;
    END_IF
END_IF

(* 快照失配只产生一个内部Z/R安全Stop事务；相关性恢复不得自动复动。 *)
IF bFastSafetyStopEvent THEN
    udiZAdapterCommandId := udiZAdapterCommandId + 1;
    IF udiZAdapterCommandId = 0 THEN
        udiZAdapterCommandId := 1;
    END_IF
    udiRAdapterCommandId := udiRAdapterCommandId + 1;
    IF udiRAdapterCommandId = 0 THEN
        udiRAdapterCommandId := 1;
    END_IF
    bNewZAdapterTransaction := TRUE;
    bNewRAdapterTransaction := TRUE;
    udiPendingZAdapterCommandId := udiZAdapterCommandId;
    udiPendingRAdapterCommandId := udiRAdapterCommandId;
    udiPendingZSequenceSourceId := 0;
    udiPendingRSequenceSourceId := 0;
    bPendingZTransactionIsSequence := FALSE;
    bPendingRTransactionIsSequence := FALSE;
    bPendingRDecelerationValid := FALSE;

    (* 使用最后一次Adapter已接受的有效减速度，构造一次纯R Stop。 *)
    stLatchedRAdapterCommand.bEnable := TRUE;
    stLatchedRAdapterCommand.bReset := FALSE;
    stLatchedRAdapterCommand.bStop := TRUE;
    stLatchedRAdapterCommand.bMoveVelocity := FALSE;
    stLatchedRAdapterCommand.rVelocity_rpm := 0.0;
    IF bLastAcceptedRDecelerationValid THEN
        stLatchedRAdapterCommand.rDeceleration_rpm_s :=
            rLastAcceptedRDeceleration_rpm_s;
    ELSE
        stLatchedRAdapterCommand.rDeceleration_rpm_s := 0.0;
    END_IF
    rPendingRDeceleration_rpm_s :=
        stLatchedRAdapterCommand.rDeceleration_rpm_s;
    bPendingRDecelerationValid := bLastAcceptedRDecelerationValid;
END_IF

(* 安全终态Reset上升沿各产生一个纯Reset事务；持续电平不重复编号。 *)
IF bSafeTerminalResetRising THEN
    udiZAdapterCommandId := udiZAdapterCommandId + 1;
    IF udiZAdapterCommandId = 0 THEN
        udiZAdapterCommandId := 1;
    END_IF
    udiRAdapterCommandId := udiRAdapterCommandId + 1;
    IF udiRAdapterCommandId = 0 THEN
        udiRAdapterCommandId := 1;
    END_IF
    bNewZAdapterTransaction := TRUE;
    bNewRAdapterTransaction := TRUE;
    udiPendingZAdapterCommandId := udiZAdapterCommandId;
    udiPendingRAdapterCommandId := udiRAdapterCommandId;
    udiPendingZSequenceSourceId := 0;
    udiPendingRSequenceSourceId := 0;
    bPendingZTransactionIsSequence := FALSE;
    bPendingRTransactionIsSequence := FALSE;
    bPendingRDecelerationValid := FALSE;

    stLatchedZSourceCommand.bEnable := FALSE;
    stLatchedZSourceCommand.bReset := TRUE;
    stLatchedZSourceCommand.bStop := FALSE;
    stLatchedZSourceCommand.bHome := FALSE;
    stLatchedZSourceCommand.bMoveAbsolute := FALSE;
    stLatchedZSourceCommand.bMoveVelocity := FALSE;
    stLatchedZSourceCommand.bUseExternalSetpoint := FALSE;
    stLatchedZSourceCommand.rHomePosition_mm := 0.0;
    stLatchedZSourceCommand.rPosition_mm := 0.0;
    stLatchedZSourceCommand.rVelocity_mm_s := 0.0;
    stLatchedZSourceCommand.rAcceleration_mm_s2 := 0.0;
    stLatchedZSourceCommand.rDeceleration_mm_s2 := 0.0;
    stLatchedZSourceCommand.eOwnerRequest := E_ZCommandOwner.Z_OWNER_NONE;

    stLatchedRAdapterCommand.bEnable := FALSE;
    stLatchedRAdapterCommand.bReset := TRUE;
    stLatchedRAdapterCommand.bStop := FALSE;
    stLatchedRAdapterCommand.bMoveVelocity := FALSE;
    stLatchedRAdapterCommand.rVelocity_rpm := 0.0;
    stLatchedRAdapterCommand.rAcceleration_rpm_s := 0.0;
    stLatchedRAdapterCommand.rDeceleration_rpm_s := 0.0;

    bFastSafetyStopLatched := FALSE;
    bHardOverridePending := FALSE;
    bHardOverrideHandled := FALSE;
    bPostResetZNormalBarrier := TRUE;
    bPostResetRNormalBarrier := TRUE;
    udiPostResetNormalBarrierRequestId :=
        GVL_FastInternal.stAcceptedCommand.nRequestId;
    bLastZSequenceSourceActive := bZSequenceSourceActive;
    bLastRSequenceSourceActive := bRSequenceSourceActive;
    udiLastZSourceCommandId := udiCurrentZSourceCommandId;
    udiLastRSourceCommandId := udiCurrentRSourceCommandId;
END_IF

stHomeCommand := stLatchedZSourceCommand;
stManualCommand := stLatchedZSourceCommand;
stApproachCommand := stLatchedZSourceCommand;
stForceProcessCommand := stLatchedZSourceCommand;
stRetractCommand := stLatchedZSourceCommand;
stHomeCommand.eOwnerRequest := E_ZCommandOwner.Z_OWNER_NONE;
stManualCommand.eOwnerRequest := E_ZCommandOwner.Z_OWNER_NONE;
stApproachCommand.eOwnerRequest := E_ZCommandOwner.Z_OWNER_NONE;
stForceProcessCommand.eOwnerRequest := E_ZCommandOwner.Z_OWNER_NONE;
stRetractCommand.eOwnerRequest := E_ZCommandOwner.Z_OWNER_NONE;
CASE stLatchedZSourceCommand.eOwnerRequest OF
    E_ZCommandOwner.Z_OWNER_HOME:
        stHomeCommand.eOwnerRequest := E_ZCommandOwner.Z_OWNER_HOME;
    E_ZCommandOwner.Z_OWNER_MANUAL:
        stManualCommand.eOwnerRequest := E_ZCommandOwner.Z_OWNER_MANUAL;
    E_ZCommandOwner.Z_OWNER_APPROACH:
        stApproachCommand.eOwnerRequest := E_ZCommandOwner.Z_OWNER_APPROACH;
    E_ZCommandOwner.Z_OWNER_FORCE_PROCESS:
        stForceProcessCommand.eOwnerRequest := E_ZCommandOwner.Z_OWNER_FORCE_PROCESS;
    E_ZCommandOwner.Z_OWNER_RETRACT:
        stRetractCommand.eOwnerRequest := E_ZCommandOwner.Z_OWNER_RETRACT;
END_CASE

bForceProcessExitComplete :=
    GVL_Status.stFast.stSequence.stMotionIntent.bForceProcessExitComplete
    AND fbZAxisExtSetpointAdapter.stStatus.bReleaseOwner;
bNormalZResetAllowed := NOT GVL_Status.stFast.stSequence.bBusy
    AND NOT bZSequenceSourceActive
    AND bExternalSafelyReleasedForReset
    AND GVL_FastInternal.stAcceptedCommand.stZAxis.bReset;
bLatchedZFaultStopRequest :=
    (stLatchedZSourceCommand.eOwnerRequest = E_ZCommandOwner.Z_OWNER_FAULT_STOP)
    OR bFastSafetyStopLatched;
stFaultStopCommand := stLatchedZSourceCommand;
fbZAxisArbiter(
    bReset := bSafeTerminalResetRising OR bNormalZResetAllowed,
    bFaultStopRequest := bLatchedZFaultStopRequest,
    stFaultStopCommand := stFaultStopCommand,
    bForceProcessExitComplete := bForceProcessExitComplete,
    stHomeCommand := stHomeCommand,
    stManualCommand := stManualCommand,
    stApproachCommand := stApproachCommand,
    stForceProcessCommand := stForceProcessCommand,
    stRetractCommand := stRetractCommand);

(* Force Ramp只使用步骤斜率与冻结Profile上限。 *)
bForceLoopRequested := GVL_Status.stFast.stSequence.bForceControlEnable
    AND bFastConfigSnapshotCurrent
    AND NOT GVL_Status.stFast.stSequence.bError
    AND NOT GVL_Status.stFast.stSequence.bAborted
    AND NOT bFastSafetyStopLatched;
rForceActual_kN := GVL_Process.stActual.fForceControlN * 0.001;
rEffectiveForceRamp_kN_s := MIN(
    GVL_Status.stFast.stSequence.rForceRamp_kN_s,
    GVL_Status.stFast.stSequence.stFastConfigSnapshot.stZForceControl.fForceRampNS
        * 0.001);
bForceRampInputValid :=
    FC_IsFiniteLReal(rValue := GVL_Status.stFast.stSequence.rForceRamp_kN_s)
    AND FC_IsFiniteLReal(rValue :=
        GVL_Status.stFast.stSequence.stFastConfigSnapshot.stZForceControl.fForceRampNS)
    AND (GVL_Status.stFast.stSequence.rForceRamp_kN_s > 0.0)
    AND (GVL_Status.stFast.stSequence.stFastConfigSnapshot.stZForceControl.fForceRampNS
        > 0.0);
IF bForceRampInputValid THEN
    rForceRampRateForFb_kN_s := rEffectiveForceRamp_kN_s;
ELSE
    rForceRampRateForFb_kN_s := -1.0;
END_IF
bForceInputsHealthy := GVL_Process.stActual.bForceValid
    AND GVL_Process.stActual.bDisplacementValid
    AND GVL_Process.stActual.bContactReferenceValid
    AND GVL_Process.stActual.bAxisSensorAgreement
    AND NOT fbZAxisNc.stStatus.bError
    AND NOT fbZAxisExtSetpointAdapter.stStatus.bError;
bFastConfigSnapshotChanged := bFastConfigSnapshotCurrent
    AND (GVL_Status.stFast.stSequence.stFastConfigSnapshot.nSequenceCommandId
        <> udiLastAppliedFastConfigCommandId);
bProfileTransferRequested := bForceLoopRequested
    AND (GVL_Status.stFast.stSequence.bForceProfileTransfer
        OR bFastConfigSnapshotChanged);

fbForceSetpointRamp(
    bEnable := bForceLoopRequested AND bForceInputsHealthy,
    bReset := bSafeTerminalReset,
    rInitialValue := rForceActual_kN,
    rTarget := GVL_Status.stFast.stSequence.rForceSet_kN,
    rRateUpPer_s := rForceRampRateForFb_kN_s,
    rRateDownPer_s := rForceRampRateForFb_kN_s,
    rCycleTime_s := rFastCycleTime_s,
    rTolerance := 0.000001);
GVL_Status.stFast.bForceSetpointRampReached := fbForceSetpointRamp.bReached;
GVL_Status.stFast.bForceSetpointRampValid := fbForceSetpointRamp.bValid;

fbZProfileSwitch(
    bEnable := bForceLoopRequested AND bForceInputsHealthy,
    bReset := bSafeTerminalReset,
    bSwitchPulse := bProfileTransferRequested,
    rPreviousVelocity_mm_s :=
        GVL_Status.stFast.stSequence.rForceTransferVelocity_mm_s,
    rVelocityFeedForward_mm_s := GVL_Status.stFast.stSequence
        .stFastConfigSnapshot.stZForceControl.fVelocityFeedForwardMmS,
    rProportionalGain_mm_s_per_kN := GVL_Status.stFast.stSequence
        .stFastConfigSnapshot.stZForceControl.fKp,
    rForceSet_kN := fbForceSetpointRamp.rOutput,
    rForceActual_kN := rForceActual_kN,
    rIntegralLimit_mm_s := GVL_Status.stFast.stSequence
        .stFastConfigSnapshot.stZForceControl.fIntegralLimit);

stZForceInput.bEnable := bForceLoopRequested AND bForceInputsHealthy
    AND NOT fbZProfileSwitch.bError;
stZForceInput.bReset := bSafeTerminalReset;
stZForceInput.bOwnerGranted := fbZAxisArbiter.eActiveOwner
    = E_ZCommandOwner.Z_OWNER_FORCE_PROCESS;
stZForceInput.bExternalActive := fbZAxisExtSetpointAdapter.stStatus.bEnabled;
stZForceInput.bForceValid := GVL_Process.stActual.bForceValid
    AND fbForceSetpointRamp.bValid;
stZForceInput.bRelativePositionValid := GVL_Process.stActual.bDisplacementValid
    AND GVL_Process.stActual.bContactReferenceValid
    AND GVL_Process.stActual.bAxisSensorAgreement;
stZForceInput.bBumplessTransfer := bProfileTransferRequested;
stZForceInput.bHardForceActive :=
    GVL_Status.stFast.stSequence.bForceHardLimitActive;
stZForceInput.bHardStrokeActive :=
    GVL_Status.stFast.stSequence.bStrokeHardLimitActive;
stZForceInput.bCollisionLimitActive :=
    GVL_Status.stFast.stSequence.bCollisionLimitActive;
stZForceInput.rForceSet_kN := GVL_Status.stFast.stSequence.rForceSet_kN;
stZForceInput.rForceActual_kN := rForceActual_kN;
stZForceInput.rRelativePosition_mm := GVL_Process.stActual.fSRelSensorMm;
stZForceInput.rTargetRelativePosition_mm :=
    GVL_Status.stFast.stSequence.rTargetRelativePosition_mm;
stZForceInput.rHardMaximumRelativePosition_mm :=
    GVL_Status.stFast.stSequence.rHardMaximumRelativePosition_mm;
stZForceInput.rTransferVelocity_mm_s :=
    GVL_Status.stFast.stSequence.rForceTransferVelocity_mm_s;
stZForceInput.rCycleTime_s := rFastCycleTime_s;
fbZForceAdmittance(
    stInput := stZForceInput,
    stProfile := GVL_Status.stFast.stSequence.stFastConfigSnapshot.stZForceControl,
    stLimits := GVL_Status.stFast.stSequence.stFastConfigSnapshot.stLimits,
    rForceSetRamped_kN := fbForceSetpointRamp.rOutput,
    bApplyIntegralPreload := fbZProfileSwitch.bAccepted,
    rIntegralPreload_mm_s := fbZProfileSwitch.rIntegralPreload_mm_s);
GVL_Status.stFast.stZForceControl := fbZForceAdmittance.stOutput;
IF fbZProfileSwitch.bAccepted THEN
    udiLastAppliedFastConfigCommandId :=
        GVL_Status.stFast.stSequence.stFastConfigSnapshot.nSequenceCommandId;
ELSIF bSafeTerminalReset THEN
    udiLastAppliedFastConfigCommandId := 0;
END_IF

(* ---------------------------------------------------------
   Hard Override跨Error/Abort保持一包精确零速Feed，直到Adapter确认接受。
   只在相关快照、ACTIVE生命周期和有效accepted基准下建立pending。
   --------------------------------------------------------- *)
bHardOverrideRequested := GVL_Status.stFast.stSequence.bForceHardLimitActive
    OR GVL_Status.stFast.stSequence.bStrokeHardLimitActive
    OR GVL_Status.stFast.stSequence.bCollisionLimitActive;
bHardOverrideAccepted := bHardOverridePending
    AND fbZAxisExtSetpointAdapter.stStatus.bFeedAccepted
    AND (fbZAxisExtSetpointAdapter.stStatus.udiFeedCycleCounter
        <> udiHardOverrideAcceptedCounter)
    AND fbZAxisExtSetpointAdapter.stStatus.bAcceptedSetpointValid
    AND (fbZAxisExtSetpointAdapter.stStatus.rAcceptedPosition_mm
        = rHardOverrideExpectedPosition_mm)
    AND (fbZAxisExtSetpointAdapter.stStatus.rAcceptedVelocity_mm_s = 0.0)
    AND (fbZAxisExtSetpointAdapter.stStatus.rAcceptedAcceleration_mm_s2 = 0.0)
    AND (fbZAxisExtSetpointAdapter.stStatus.nAcceptedDirection
        = nHardOverrideExpectedDirection);
IF bHardOverrideAccepted THEN
    bHardOverridePending := FALSE;
    bHardOverrideHandled := TRUE;
END_IF
IF bSafeTerminalResetRising THEN
    bHardOverridePending := FALSE;
    bHardOverrideHandled := FALSE;
ELSIF NOT bHardOverrideRequested AND NOT bHardOverridePending THEN
    bHardOverrideHandled := FALSE;
END_IF
bHardOverrideStart := bFastConfigSnapshotCurrent
    AND NOT bFastSafetyStopLatched
    AND (fbZAxisExtSetpointAdapter.stStatus.eState
        = E_ZExtSetpointState.Z_EXT_ACTIVE)
    AND fbZAxisExtSetpointAdapter.stStatus.bAcceptedSetpointValid
    AND bHardOverrideRequested
    AND NOT bHardOverridePending
    AND NOT bHardOverrideHandled
    AND ((fbZAxisExtSetpointAdapter.stStatus.rAcceptedVelocity_mm_s > 0.0)
        OR (fbZExternalTrajectory.stOutput.rVelocity_mm_s > 0.0));
IF bHardOverrideStart THEN
    bHardOverridePending := TRUE;
    rHardOverrideExpectedPosition_mm :=
        fbZAxisExtSetpointAdapter.stStatus.rAcceptedPosition_mm;
    nHardOverrideExpectedDirection :=
        fbZAxisExtSetpointAdapter.stStatus.nAcceptedDirection;
    udiHardOverrideAcceptedCounter :=
        fbZAxisExtSetpointAdapter.stStatus.udiFeedCycleCounter;
END_IF

(* External轨迹只读Adapter accepted状态和同一冻结快照。 *)
IF GVL_Status.stFast.stSequence.bForceControlEnable THEN
    rTrajectoryTargetVelocity_mm_s :=
        fbZForceAdmittance.stOutput.rVelocityCommand_mm_s;
ELSE
    rTrajectoryTargetVelocity_mm_s := GVL_Status.stFast.stSequence
        .stMotionIntent.rExternalTargetVelocity_mm_s;
END_IF
stTrajectoryInput.bEnable := (bFastConfigSnapshotCurrent
        AND NOT GVL_Status.stFast.stSequence.bError
        AND NOT GVL_Status.stFast.stSequence.bAborted
        AND NOT bFastSafetyStopLatched)
    OR (bHardOverridePending
        AND bFastConfigSnapshotCurrent
        AND NOT bFastSafetyStopLatched);
stTrajectoryInput.bReset := bSafeTerminalReset;
stTrajectoryInput.eExternalState := fbZAxisExtSetpointAdapter.stStatus.eState;
stTrajectoryInput.bAcceptedSetpointValid :=
    fbZAxisExtSetpointAdapter.stStatus.bAcceptedSetpointValid;
stTrajectoryInput.bFeedAccepted :=
    fbZAxisExtSetpointAdapter.stStatus.bFeedAccepted;
stTrajectoryInput.udiAcceptedFeedCycleCounter :=
    fbZAxisExtSetpointAdapter.stStatus.udiFeedCycleCounter;
stTrajectoryInput.rAcceptedPosition_mm :=
    fbZAxisExtSetpointAdapter.stStatus.rAcceptedPosition_mm;
stTrajectoryInput.rAcceptedVelocity_mm_s :=
    fbZAxisExtSetpointAdapter.stStatus.rAcceptedVelocity_mm_s;
stTrajectoryInput.rAcceptedAcceleration_mm_s2 :=
    fbZAxisExtSetpointAdapter.stStatus.rAcceptedAcceleration_mm_s2;
stTrajectoryInput.nAcceptedDirection :=
    fbZAxisExtSetpointAdapter.stStatus.nAcceptedDirection;
stTrajectoryInput.bInhibitPositiveMotion :=
    GVL_Status.stFast.stSequence.bForceHardLimitActive
    OR GVL_Status.stFast.stSequence.bStrokeHardLimitActive
    OR GVL_Status.stFast.stSequence.bCollisionLimitActive
    OR bHardOverridePending;
stTrajectoryInput.rTargetVelocity_mm_s := rTrajectoryTargetVelocity_mm_s;
stTrajectoryInput.rCycleTime_s := rFastCycleTime_s;
stTrajectoryInput.rMinimumPosition_mm :=
    GVL_Status.stFast.stSequence.stFastConfigSnapshot.stLimits.fZMinPositionMm;
stTrajectoryInput.rMaximumPosition_mm :=
    GVL_Status.stFast.stSequence.stFastConfigSnapshot.stLimits.fZMaxPositionMm;
stTrajectoryInput.rMaximumVelocity_mm_s :=
    GVL_Status.stFast.stSequence.stFastConfigSnapshot.stLimits.fZMaxVelocityMmS;
stTrajectoryInput.rMaximumAcceleration_mm_s2 :=
    GVL_Status.stFast.stSequence.stFastConfigSnapshot.stLimits.fZMaxAccelerationMmS2;
stTrajectoryInput.rStandstillVelocity_mm_s := GVL_Status.stFast.stSequence
    .stFastConfigSnapshot.stZExtSetpoint.rStandstillVelocity_mm_s;
stTrajectoryInput.rMaximumPositionDeviation_mm := GVL_Status.stFast.stSequence
    .stFastConfigSnapshot.stZExtSetpoint.rMaximumPositionDeviation_mm;
stTrajectoryInput.nDirectionHoldCycles := GVL_Status.stFast.stSequence
    .stFastConfigSnapshot.stZExtSetpoint.nDirectionHoldCycles;
fbZExternalTrajectory(stInput := stTrajectoryInput);
GVL_Status.stFast.stZExternalTrajectory := fbZExternalTrajectory.stOutput;
bHardOverridePackageExact := bHardOverridePending
    AND bFastConfigSnapshotCurrent
    AND NOT bFastSafetyStopLatched
    AND fbZExternalTrajectory.stOutput.bActive
    AND NOT fbZExternalTrajectory.stOutput.bFault
    AND fbZExternalTrajectory.stOutput.bPositiveMotionInhibited
    AND (fbZExternalTrajectory.stOutput.rPosition_mm
        = rHardOverrideExpectedPosition_mm)
    AND (fbZExternalTrajectory.stOutput.rVelocity_mm_s = 0.0)
    AND (fbZExternalTrajectory.stOutput.rAcceleration_mm_s2 = 0.0)
    AND (fbZExternalTrajectory.stOutput.nDirection
        = nHardOverrideExpectedDirection);

stExtCommand.bReset := bSafeTerminalResetRising;
stExtCommand.bEnable :=
    GVL_Status.stFast.stSequence.stMotionIntent.bExternalEnableRequest;
stExtCommand.bFeed := fbZExternalTrajectory.stOutput.bActive
    AND NOT fbZExternalTrajectory.stOutput.bFault;
stExtCommand.bDisable :=
    GVL_Status.stFast.stSequence.stMotionIntent.bExternalDisableRequest
    OR fbZExternalTrajectory.stOutput.bFault;
stExtCommand.bPositiveMotionInhibit :=
    fbZExternalTrajectory.stOutput.bPositiveMotionInhibited;
stExtCommand.rPosition_mm := fbZExternalTrajectory.stOutput.rPosition_mm;
stExtCommand.rVelocity_mm_s := fbZExternalTrajectory.stOutput.rVelocity_mm_s;
stExtCommand.rAcceleration_mm_s2 :=
    fbZExternalTrajectory.stOutput.rAcceleration_mm_s2;
stExtCommand.nDirection := fbZExternalTrajectory.stOutput.nDirection;

bFastPathSafetyExit := NOT bFastConfigSnapshotCurrent
    OR bFastSafetyStopLatched
    OR GVL_Status.stFast.stSequence.bError
    OR GVL_Status.stFast.stSequence.bAborted
    OR fbZProfileSwitch.bError
    OR (bForceLoopRequested AND NOT fbForceSetpointRamp.bValid)
    OR (GVL_Status.stFast.stSequence.bForceControlEnable
        AND (NOT bForceInputsHealthy OR fbZForceAdmittance.stOutput.bFault));
IF bFastPathSafetyExit THEN
    stExtCommand.bEnable := FALSE;
    stExtCommand.bFeed := FALSE;
    stExtCommand.bDisable := TRUE;
END_IF

(* Error/Abort不能吞掉已建立的硬覆盖包；仅精确包保留marker和Feed。 *)
IF bHardOverrideHandled AND bHardOverrideRequested THEN
    stExtCommand.bEnable := FALSE;
    stExtCommand.bFeed := FALSE;
    stExtCommand.bDisable := TRUE;
    stExtCommand.bPositiveMotionInhibit := FALSE;
END_IF
IF bHardOverridePending THEN
    stExtCommand.bFeed := bHardOverridePackageExact;
    stExtCommand.bDisable := TRUE;
    stExtCommand.bPositiveMotionInhibit := bHardOverridePackageExact;
END_IF
IF NOT stExtCommand.bFeed THEN
    (* Feed FALSE时绝不把marker送进Adapter的硬覆盖优先分支。 *)
    stExtCommand.bPositiveMotionInhibit := FALSE;
END_IF

(* 标准Z Adapter在External通道释放前冻结事务号。 *)
stSelectedZCommand := fbZAxisArbiter.stCommand;
stSelectedZCommand.bReset := bNormalZResetAllowed OR bSafeTerminalResetRising;
bExternalCommandChannelBusy := (fbZAxisExtSetpointAdapter.stStatus.eState
    <> E_ZExtSetpointState.Z_EXT_IDLE)
    AND NOT fbZAxisExtSetpointAdapter.stStatus.bReleaseOwner;
IF bExternalCommandChannelBusy THEN
    stSelectedZCommand.bEnable := TRUE;
    stSelectedZCommand.bReset := FALSE;
    stSelectedZCommand.bStop := FALSE;
    stSelectedZCommand.bHome := FALSE;
    stSelectedZCommand.bMoveAbsolute := FALSE;
    stSelectedZCommand.bMoveVelocity := FALSE;
    stSelectedZCommand.bUseExternalSetpoint := TRUE;
    udiZStandardCommandId := fbZAxisNc.udiAcceptedCommandId;
ELSE
    udiZStandardCommandId := udiZAdapterCommandId;
END_IF
fbZAxisNc(
    Axis := GVL_IO.Z_axis,
    bDriveLinked := GVL_Status.stHardwareBinding.bZAxisDriveLinked,
    udiCommandId := udiZStandardCommandId,
    stCommand := stSelectedZCommand);
GVL_Status.stFast.stZAxis := fbZAxisNc.stStatus;
IF bPendingZTransactionIsSequence
    AND (fbZAxisNc.udiAcceptedCommandId = udiPendingZAdapterCommandId)
    AND (udiPendingZSequenceSourceId <> 0) THEN
    udiAcceptedZSequenceSourceId := udiPendingZSequenceSourceId;
    GVL_Status.stFast.udiAcceptedSequenceZCommandId :=
        udiPendingZSequenceSourceId;
END_IF

fbZAxisExtSetpointAdapter(
    Axis := GVL_IO.Z_axis,
    bDriveLinked := GVL_Status.stHardwareBinding.bZAxisDriveLinked,
    bOwnerGranted := fbZAxisArbiter.eActiveOwner
        = E_ZCommandOwner.Z_OWNER_FORCE_PROCESS,
    bLimitsValid := GVL_Status.stFast.stSequence
        .stFastConfigSnapshot.stLimits.bValid,
    bAxisReady := fbZAxisNc.stStatus.bReady,
    bAxisError := fbZAxisNc.stStatus.bError,
    rCycleTime_s := rFastCycleTime_s,
    rMinimumPosition_mm := GVL_Status.stFast.stSequence
        .stFastConfigSnapshot.stLimits.fZMinPositionMm,
    rMaximumPosition_mm := GVL_Status.stFast.stSequence
        .stFastConfigSnapshot.stLimits.fZMaxPositionMm,
    rMaximumVelocity_mm_s := GVL_Status.stFast.stSequence
        .stFastConfigSnapshot.stLimits.fZMaxVelocityMmS,
    rMaximumAcceleration_mm_s2 := GVL_Status.stFast.stSequence
        .stFastConfigSnapshot.stLimits.fZMaxAccelerationMmS2,
    stConfig := GVL_Status.stFast.stSequence
        .stFastConfigSnapshot.stZExtSetpoint,
    stCommand := stExtCommand);
GVL_Status.stFast.stZExtSetpoint := fbZAxisExtSetpointAdapter.stStatus;
GVL_Status.stFast.stZAxis.bExternalSetpointActive :=
    fbZAxisExtSetpointAdapter.stStatus.bEnabled;
GVL_Status.stFast.stZAxis.eActiveOwner := fbZAxisArbiter.eActiveOwner;
IF fbZAxisExtSetpointAdapter.stStatus.bError THEN
    GVL_Status.stFast.stZAxis.bError := TRUE;
    GVL_Status.stFast.stZAxis.nErrorId :=
        fbZAxisExtSetpointAdapter.stStatus.nErrorId;
END_IF

(* R源路由：源切换或同源更新仅创建一次Adapter事务。 *)
bRNormalSourceBlockedByReset := bPostResetRNormalBarrier
    AND NOT bAcceptedFastPackageNewerThanReset;
bNewRSourceTransaction := (udiCurrentRSourceCommandId <> 0)
    AND ((bRSequenceSourceActive <> bLastRSequenceSourceActive)
        OR FC_IsNewerRequestId(
            udiCandidate := udiCurrentRSourceCommandId,
            udiReference := udiLastRSourceCommandId));
IF bRNormalSourceBlockedByReset THEN
    bNewRSourceTransaction := FALSE;
END_IF
IF NOT bFastSafetyStopLatched AND NOT bSafeTerminalResetRising THEN
    bNewRAdapterTransaction := bNewRSourceTransaction;
END_IF
IF bNewRAdapterTransaction THEN
IF NOT bFastSafetyStopLatched AND NOT bSafeTerminalResetRising THEN
    udiRAdapterCommandId := udiRAdapterCommandId + 1;
    IF udiRAdapterCommandId = 0 THEN
        udiRAdapterCommandId := 1;
    END_IF
    udiLastRSourceCommandId := udiCurrentRSourceCommandId;
    stLatchedRAdapterCommand := stCandidateRSourceCommand;
    bLastRSequenceSourceActive := bRSequenceSourceActive;
    udiPendingRAdapterCommandId := udiRAdapterCommandId;
    rPendingRDeceleration_rpm_s :=
        stCandidateRSourceCommand.rDeceleration_rpm_s;
    bPendingRDecelerationValid := FC_IsFiniteLReal(
        rValue := rPendingRDeceleration_rpm_s)
        AND (rPendingRDeceleration_rpm_s > 0.0);
    bPendingRTransactionIsSequence := bRSequenceSourceActive;
    IF bRSequenceSourceActive THEN
        udiPendingRSequenceSourceId := udiCurrentSequenceRSourceId;
    ELSE
        udiPendingRSequenceSourceId := 0;
    END_IF
    IF bPostResetRNormalBarrier
        AND NOT bRSequenceSourceActive
        AND bAcceptedFastPackageNewerThanReset THEN
        bPostResetRNormalBarrier := FALSE;
    END_IF
END_IF
END_IF
stSelectedRCommand := stLatchedRAdapterCommand;

bRSpeedRampSafeReset := bSafeTerminalReset
    AND NOT bRSequenceSourceActive
    AND GVL_Status.stFast.stRAxis.bStandstill;
fbRSpeedRamp(
    bEnable := bRSequenceSourceActive OR stSelectedRCommand.bEnable,
    bReset := bNewRAdapterTransaction OR bRSpeedRampSafeReset,
    rInitialValue := GVL_Status.stFast.stRAxis.rActualVelocity_rpm,
    rTarget := stSelectedRCommand.rVelocity_rpm,
    rRateUpPer_s := stSelectedRCommand.rAcceleration_rpm_s,
    rRateDownPer_s := stSelectedRCommand.rDeceleration_rpm_s,
    rCycleTime_s := rFastCycleTime_s,
    rTolerance := 0.0);
GVL_Status.stFast.rRSpeedEnvelope_rpm := fbRSpeedRamp.rOutput;
GVL_Status.stFast.bRSpeedRampBusy := fbRSpeedRamp.bBusy;
GVL_Status.stFast.bRSpeedRampReached := fbRSpeedRamp.bReached;
GVL_Status.stFast.bRSpeedRampValid := fbRSpeedRamp.bValid;

fbRAxisNc(
    Axis := GVL_IO.R_axis,
    bDriveLinked := GVL_Status.stHardwareBinding.bRAxisDriveLinked,
    udiCommandId := udiRAdapterCommandId,
    stCommand := stSelectedRCommand);
GVL_Status.stFast.stRAxis := fbRAxisNc.stStatus;
IF bPendingRTransactionIsSequence
    AND (fbRAxisNc.udiAcceptedCommandId = udiPendingRAdapterCommandId)
    AND (udiPendingRSequenceSourceId <> 0) THEN
    udiAcceptedRSequenceSourceId := udiPendingRSequenceSourceId;
    GVL_Status.stFast.udiAcceptedSequenceRCommandId :=
        udiPendingRSequenceSourceId;
END_IF

(* 固定报警槽：External/轨迹=7，Force算法/Profile=8。 *)
GVL_Alarm.astRequests[7].eCode := E_AlarmCode.ALARM_EXTERNAL_SETPOINT_FAULT;
GVL_Alarm.astRequests[7].eLevel := E_AlarmLevel.ALARM_LEVEL_FAULT;
GVL_Alarm.astRequests[7].nTextId := 2200;
GVL_Alarm.astRequests[7].nSourceId := 7;
GVL_Alarm.astRequests[7].bLatch := TRUE;
GVL_Alarm.astRequests[7].bActive :=
    fbZAxisExtSetpointAdapter.stStatus.bError
    OR fbZExternalTrajectory.stOutput.bFault;
GVL_Alarm.astRequests[8].eCode := E_AlarmCode.ALARM_FORCE_CONTROL_FAULT;
GVL_Alarm.astRequests[8].eLevel := E_AlarmLevel.ALARM_LEVEL_FAULT;
GVL_Alarm.astRequests[8].nTextId := 2500;
GVL_Alarm.astRequests[8].nSourceId := 8;
GVL_Alarm.astRequests[8].bLatch := TRUE;
GVL_Alarm.astRequests[8].bActive := fbZForceAdmittance.stOutput.bFault
    OR fbZProfileSwitch.bError;

GVL_Status.stFast.nAcceptedRequestId :=
    GVL_FastInternal.stAcceptedCommand.nRequestId;

END_PROGRAM

// ---- POUs/FunctionBlocks/Axis/FB_AxisCommandArbiter.TcPOU
FUNCTION_BLOCK FB_AxisCommandArbiter
VAR_INPUT
    (* 复位Owner和已选命令。 *)
    bReset : BOOL;
    (* 最高优先级故障受控停止请求。 *)
    bFaultStopRequest : BOOL;
    stFaultStopCommand : ST_ZAxisCommand;
    (* 力过程已完成受控退出，允许转交Owner。 *)
    bForceProcessExitComplete : BOOL;
    (* 回零Owner候选命令。 *)
    stHomeCommand : ST_ZAxisCommand;
    (* 手动Owner候选命令。 *)
    stManualCommand : ST_ZAxisCommand;
    (* 接近Owner候选命令。 *)
    stApproachCommand : ST_ZAxisCommand;
    (* 力过程Owner候选命令。 *)
    stForceProcessCommand : ST_ZAxisCommand;
    (* 回撤Owner候选命令。 *)
    stRetractCommand : ST_ZAxisCommand;
END_VAR
VAR_OUTPUT
    (* 唯一获准发往Z轴Adapter的命令。 *)
    stCommand : ST_ZAxisCommand;
    (* 当前唯一Z轴命令Owner。 *)
    eActiveOwner : E_ZCommandOwner;
    (* 当前扫描存在有效Owner。 *)
    bOwnerActive : BOOL;
    (* 力过程尚未受控退出，Owner切换被拒绝。 *)
    bTransitionDenied : BOOL;
END_VAR
VAR
    (* 力过程候选在当前扫描有效。 *)
    bForceProcessRequested : BOOL;
END_VAR

(* ---------------------------------------------------------
   Z轴命令Owner仲裁状态。
   进入：Task_CffFast每扫描调用。
   动作：Fault Stop最高；活动力过程须先完成受控退出；其后
         按Home、Retract、Approach、Manual选择唯一命令。
   成功：只发布一个ST_ZAxisCommand和一个ActiveOwner。
   超时：由上层流程负责；本FB不访问任务时钟或硬件。
   Fault：立即选择FAULT_STOP并发布受控Stop。
   --------------------------------------------------------- *)
bForceProcessRequested := stForceProcessCommand.eOwnerRequest = E_ZCommandOwner.Z_OWNER_FORCE_PROCESS;
bTransitionDenied := FALSE;

IF bReset THEN
    eActiveOwner := E_ZCommandOwner.Z_OWNER_NONE;
ELSIF bFaultStopRequest THEN
    eActiveOwner := E_ZCommandOwner.Z_OWNER_FAULT_STOP;
ELSIF (eActiveOwner = E_ZCommandOwner.Z_OWNER_FORCE_PROCESS)
    AND NOT bForceProcessExitComplete THEN
    eActiveOwner := E_ZCommandOwner.Z_OWNER_FORCE_PROCESS;
    bTransitionDenied := NOT bForceProcessRequested;
ELSIF bForceProcessRequested THEN
    eActiveOwner := E_ZCommandOwner.Z_OWNER_FORCE_PROCESS;
ELSIF stHomeCommand.eOwnerRequest = E_ZCommandOwner.Z_OWNER_HOME THEN
    eActiveOwner := E_ZCommandOwner.Z_OWNER_HOME;
ELSIF stRetractCommand.eOwnerRequest = E_ZCommandOwner.Z_OWNER_RETRACT THEN
    eActiveOwner := E_ZCommandOwner.Z_OWNER_RETRACT;
ELSIF stApproachCommand.eOwnerRequest = E_ZCommandOwner.Z_OWNER_APPROACH THEN
    eActiveOwner := E_ZCommandOwner.Z_OWNER_APPROACH;
ELSIF stManualCommand.eOwnerRequest = E_ZCommandOwner.Z_OWNER_MANUAL THEN
    eActiveOwner := E_ZCommandOwner.Z_OWNER_MANUAL;
ELSE
    eActiveOwner := E_ZCommandOwner.Z_OWNER_NONE;
END_IF

CASE eActiveOwner OF
    E_ZCommandOwner.Z_OWNER_HOME:
        stCommand := stHomeCommand;
    E_ZCommandOwner.Z_OWNER_MANUAL:
        stCommand := stManualCommand;
    E_ZCommandOwner.Z_OWNER_APPROACH:
        stCommand := stApproachCommand;
    E_ZCommandOwner.Z_OWNER_FORCE_PROCESS:
        IF bForceProcessRequested THEN
            stCommand := stForceProcessCommand;
        END_IF
    E_ZCommandOwner.Z_OWNER_RETRACT:
        stCommand := stRetractCommand;
    E_ZCommandOwner.Z_OWNER_FAULT_STOP:
        stCommand := stFaultStopCommand;
        stCommand.bEnable := TRUE;
        stCommand.bReset := FALSE;
        stCommand.bStop := TRUE;
        stCommand.bHome := FALSE;
        stCommand.bMoveAbsolute := FALSE;
        stCommand.bMoveVelocity := FALSE;
        stCommand.bUseExternalSetpoint := FALSE;
        stCommand.rHomePosition_mm := 0.0;
        stCommand.rPosition_mm := 0.0;
        stCommand.rVelocity_mm_s := 0.0;
        stCommand.rAcceleration_mm_s2 := 0.0;
        stCommand.eOwnerRequest := E_ZCommandOwner.Z_OWNER_FAULT_STOP;
    ELSE
        stCommand.bEnable := FALSE;
        stCommand.bReset := FALSE;
        stCommand.bStop := FALSE;
        stCommand.bHome := FALSE;
        stCommand.bMoveAbsolute := FALSE;
        stCommand.bMoveVelocity := FALSE;
        stCommand.bUseExternalSetpoint := FALSE;
        stCommand.rHomePosition_mm := 0.0;
        stCommand.rPosition_mm := 0.0;
        stCommand.rVelocity_mm_s := 0.0;
        stCommand.rAcceleration_mm_s2 := 0.0;
        stCommand.rDeceleration_mm_s2 := 0.0;
        stCommand.eOwnerRequest := E_ZCommandOwner.Z_OWNER_NONE;
END_CASE

bOwnerActive := eActiveOwner <> E_ZCommandOwner.Z_OWNER_NONE;

END_FUNCTION_BLOCK

// ---- POUs/FunctionBlocks/Utility/FB_SetpointRamp.TcPOU
FUNCTION_BLOCK FB_SetpointRamp
VAR_INPUT
    (* 斜坡运行许可。 *)
    bEnable : BOOL;
    (* 内部状态复位请求。 *)
    bReset : BOOL;
    (* 首次使能或复位后的连续起始值。 *)
    rInitialValue : LREAL;
    (* 需要平滑到达的目标值。 *)
    rTarget : LREAL;
    (* 正方向最大变化率，单位每秒。 *)
    rRateUpPer_s : LREAL;
    (* 负方向最大变化率绝对值，单位每秒。 *)
    rRateDownPer_s : LREAL;
    (* 实际调用周期，单位秒。 *)
    rCycleTime_s : LREAL;
    (* 判断到达目标的绝对容差。 *)
    rTolerance : LREAL;
END_VAR
VAR_OUTPUT
    (* 当前斜坡输出。 *)
    rOutput : LREAL;
    (* 仍在向目标变化时为TRUE。 *)
    bBusy : BOOL;
    (* 输出进入目标容差且不再需要变化时为TRUE。 *)
    bReached : BOOL;
    (* 周期、速率和输入均有效时为TRUE。 *)
    bValid : BOOL;
END_VAR
VAR
    (* 已用起始值建立连续输出。 *)
    bInitialized : BOOL;
    (* 所有可能影响输出的参数均有限且位于允许符号范围。 *)
    bInputsValid : BOOL;
    (* 非负到达容差。 *)
    rAbsoluteTolerance : LREAL;
END_VAR

bInputsValid := (rCycleTime_s > 0.0)
    AND (rRateUpPer_s >= 0.0)
    AND (rRateDownPer_s >= 0.0)
    AND (rTolerance >= 0.0)
    AND FC_IsFiniteLReal(rValue := rInitialValue)
    AND FC_IsFiniteLReal(rValue := rTarget)
    AND FC_IsFiniteLReal(rValue := rRateUpPer_s)
    AND FC_IsFiniteLReal(rValue := rRateDownPer_s)
    AND FC_IsFiniteLReal(rValue := rCycleTime_s)
    AND FC_IsFiniteLReal(rValue := rTolerance);

IF bReset OR NOT bEnable THEN
    IF bInputsValid THEN
        rOutput := rInitialValue;
    END_IF
    bInitialized := bEnable AND bInputsValid;
    bBusy := FALSE;
    bReached := FALSE;
    bValid := FALSE;
    IF NOT bEnable OR NOT bInputsValid THEN
        RETURN;
    END_IF
END_IF

bValid := bInputsValid;
IF NOT bValid THEN
    (* 参数无效时保持最后连续输出，不向设备发布跳变。 *)
    bBusy := FALSE;
    bReached := FALSE;
    RETURN;
END_IF

IF NOT bInitialized THEN
    rOutput := rInitialValue;
    bInitialized := TRUE;
END_IF

rOutput := FC_LimitRate(
    rCurrent := rOutput,
    rTarget := rTarget,
    rRateUpPer_s := rRateUpPer_s,
    rRateDownPer_s := rRateDownPer_s,
    rCycleTime_s := rCycleTime_s);
rAbsoluteTolerance := rTolerance;
bReached := ABS(rTarget - rOutput) <= rAbsoluteTolerance;
bBusy := NOT bReached;

END_FUNCTION_BLOCK

// ---- POUs/Functions/FC_LimitRate.TcPOU
FUNCTION FC_LimitRate : LREAL
VAR_INPUT
    (* 当前输出值。 *)
    rCurrent : LREAL;
    (* 本周期目标值。 *)
    rTarget : LREAL;
    (* 正方向最大变化率，单位每秒，必须非负。 *)
    rRateUpPer_s : LREAL;
    (* 负方向最大变化率绝对值，单位每秒，必须非负。 *)
    rRateDownPer_s : LREAL;
    (* 实际调用周期，单位秒。 *)
    rCycleTime_s : LREAL;
END_VAR
VAR
    (* 本周期允许的正向增量。 *)
    rMaximumUpStep : LREAL;
    (* 本周期允许的负向增量绝对值。 *)
    rMaximumDownStep : LREAL;
    (* 目标与当前值之差。 *)
    rDelta : LREAL;
END_VAR

(* 无效周期或负速率时保持当前值，防止产生方向相反的跳变。 *)
IF (rCycleTime_s <= 0.0) OR (rRateUpPer_s < 0.0) OR (rRateDownPer_s < 0.0)
    OR NOT FC_IsFiniteLReal(rValue := rCurrent)
    OR NOT FC_IsFiniteLReal(rValue := rTarget)
    OR NOT FC_IsFiniteLReal(rValue := rRateUpPer_s)
    OR NOT FC_IsFiniteLReal(rValue := rRateDownPer_s) THEN
    FC_LimitRate := rCurrent;
    RETURN;
END_IF

rMaximumUpStep := rRateUpPer_s * rCycleTime_s;
rMaximumDownStep := rRateDownPer_s * rCycleTime_s;
rDelta := rTarget - rCurrent;

IF rDelta > rMaximumUpStep THEN
    FC_LimitRate := rCurrent + rMaximumUpStep;
ELSIF rDelta < -rMaximumDownStep THEN
    FC_LimitRate := rCurrent - rMaximumDownStep;
ELSE
    FC_LimitRate := rTarget;
END_IF

END_FUNCTION

// ---- POUs/FunctionBlocks/Control/FB_BumplessProfileSwitch.TcPOU
FUNCTION_BLOCK FB_BumplessProfileSwitch
VAR_INPUT
    (* 无扰计算许可；FALSE时清除脉冲历史和输出状态。 *)
    bEnable : BOOL;
    (* 清除脉冲历史、接受状态和积分预置。 *)
    bReset : BOOL;
    (* Contact接管或Profile变化的单扫描请求。 *)
    bSwitchPulse : BOOL;
    (* 切换前连续速度命令，向下为正，单位mm/s。 *)
    rPreviousVelocity_mm_s : LREAL;
    (* 新Profile速度前馈，向下为正，单位mm/s。 *)
    rVelocityFeedForward_mm_s : LREAL;
    (* 新Profile比例增益，单位mm/s/kN。 *)
    rProportionalGain_mm_s_per_kN : LREAL;
    (* 新Profile起始目标力，单位kN。 *)
    rForceSet_kN : LREAL;
    (* 当前ForceControl实际力，单位kN。 *)
    rForceActual_kN : LREAL;
    (* 新Profile积分项绝对限幅，单位mm/s。 *)
    rIntegralLimit_mm_s : LREAL;
END_VAR
VAR_OUTPUT
    (* 限幅后的新积分初值，单位mm/s。 *)
    rIntegralPreload_mm_s : LREAL;
    (* 当前扫描成功接受一个切换上升沿。 *)
    bAccepted : BOOL;
    (* 全部输入有限且参数范围有效。 *)
    bValid : BOOL;
    (* 切换脉冲到来时输入无效。 *)
    bError : BOOL;
    (* 确定性的无扰切换错误编号，0表示无错误。 *)
    nErrorId : UDINT;
END_VAR
VAR
    (* 上一扫描的切换请求，用于只接受上升沿。 *)
    bPreviousSwitchPulse : BOOL;
    (* 当前扫描检测到切换上升沿。 *)
    bSwitchRise : BOOL;
    (* 限幅前的积分预置，单位mm/s。 *)
    rRawIntegralPreload_mm_s : LREAL;
END_VAR

IF bReset THEN
    rIntegralPreload_mm_s := 0.0;
    bAccepted := FALSE;
    bValid := FALSE;
    bError := FALSE;
    nErrorId := 0;
    bPreviousSwitchPulse := FALSE;
    RETURN;
END_IF

bAccepted := FALSE;
IF NOT bEnable THEN
    bValid := FALSE;
    bPreviousSwitchPulse := FALSE;
    RETURN;
END_IF

IF bError THEN
    (* 无效无扰预置必须由显式Reset清除，禁止下一扫描自动恢复。 *)
    RETURN;
END_IF

bSwitchRise := bSwitchPulse AND NOT bPreviousSwitchPulse;
bPreviousSwitchPulse := bSwitchPulse;

bValid := FC_IsFiniteLReal(rValue := rPreviousVelocity_mm_s)
    AND FC_IsFiniteLReal(rValue := rVelocityFeedForward_mm_s)
    AND FC_IsFiniteLReal(rValue := rProportionalGain_mm_s_per_kN)
    AND FC_IsFiniteLReal(rValue := rForceSet_kN)
    AND FC_IsFiniteLReal(rValue := rForceActual_kN)
    AND FC_IsFiniteLReal(rValue := rIntegralLimit_mm_s)
    AND (rProportionalGain_mm_s_per_kN >= 0.0)
    AND (rIntegralLimit_mm_s >= 0.0);

IF bSwitchRise THEN
    IF NOT bValid THEN
        bError := TRUE;
        nErrorId := 16#00008001;
    ELSE
        (* 用新Profile重算积分，使切换前后速度命令连续。 *)
        rRawIntegralPreload_mm_s := rPreviousVelocity_mm_s
            - rVelocityFeedForward_mm_s
            - rProportionalGain_mm_s_per_kN * (rForceSet_kN - rForceActual_kN);
        IF NOT FC_IsFiniteLReal(rValue := rRawIntegralPreload_mm_s) THEN
            bError := TRUE;
            nErrorId := 16#00008002;
        ELSE
            rIntegralPreload_mm_s := FC_ClampLReal(
                rValue := rRawIntegralPreload_mm_s,
                rMinimum := -ABS(rIntegralLimit_mm_s),
                rMaximum := ABS(rIntegralLimit_mm_s));
            IF NOT FC_IsFiniteLReal(rValue := rIntegralPreload_mm_s) THEN
                bError := TRUE;
                nErrorId := 16#00008003;
            ELSE
                bAccepted := TRUE;
                bError := FALSE;
                nErrorId := 0;
            END_IF
        END_IF
    END_IF
END_IF

END_FUNCTION_BLOCK

// ---- POUs/FunctionBlocks/Control/FB_ZForceAdmittance.TcPOU
FUNCTION_BLOCK FB_ZForceAdmittance
VAR_INPUT
    (* 调用者完整赋值的力控、有效性和硬边界输入。 *)
    stInput : ST_ZForceControlInput;
    (* 候选导纳Profile；只有无扰预置成功后才提交。 *)
    stProfile : ST_ZForceControlProfile;
    (* 当前机器硬限值；FB不访问全局配置。 *)
    stLimits : ST_MachineLimits;
    (* 已由独立Ramp生成的连续目标力，单位kN。 *)
    rForceSetRamped_kN : LREAL;
    (* 当前扫描应用无扰切换FB生成的积分预置。 *)
    bApplyIntegralPreload : BOOL;
    (* 无扰切换后的积分初值，单位mm/s。 *)
    rIntegralPreload_mm_s : LREAL;
END_VAR
VAR_OUTPUT
    (* 导纳速度和完整诊断输出。 *)
    stOutput : ST_ZForceControlOutput;
END_VAR
VAR
    (* 最近一次完成无扰预置并提交的Profile快照。 *)
    stAppliedProfile : ST_ZForceControlProfile;
    (* 与Profile同一次无扰提交的Z轴/过程机器限值快照。 *)
    stAppliedLimits : ST_MachineLimits;
    (* 当前Enable生命周期已经提交一个Profile。 *)
    bProfileInitialized : BOOL;
    (* 候选Profile或几何目标绕过无扰切换。 *)
    bProfileMismatch : BOOL;
    (* 机器限值在未提交新Profile时发生变化。 *)
    bLimitsMismatch : BOOL;
    (* 算法故障锁存；只有显式Reset清除。 *)
    bFaultLatched : BOOL;
    (* 已锁存的确定性故障编号。 *)
    udiLatchedFaultId : UDINT;
    (* Profile、机器限值和周期均满足算法运行条件。 *)
    bConfigurationValid : BOOL;
    (* 本周期所有工艺输入均为有限数。 *)
    bInputFinite : BOOL;
    (* Hard Force、Hard S_rel或Collision边界当前有效。 *)
    bHardLimitActive : BOOL;
    (* 向下硬边界当前有效，但不禁止受控上抬。 *)
    bDownwardBoundaryActive : BOOL;
    (* 当前周期冻结积分。 *)
    bFreezeIntegral : BOOL;
    (* 当前力误差要求继续向下。 *)
    bErrorRequestsDownward : BOOL;
    (* Rate Limit后的速度超过当前S_rel制动包络。 *)
    bEnvelopeViolation : BOOL;
    (* PI积分分量，单位mm/s。 *)
    rIntegralTerm_mm_s : LREAL;
    (* 本周期限幅前的积分更新候选，单位mm/s。 *)
    rUpdatedIntegralTerm_mm_s : LREAL;
    (* 力误差，单位kN。 *)
    rForceError_kN : LREAL;
    (* 未饱和PI速度，单位mm/s。 *)
    rUnsaturatedVelocity_mm_s : LREAL;
    (* 固定硬边界限幅后的速度，单位mm/s。 *)
    rBoundaryLimitedVelocity_mm_s : LREAL;
    (* 包含加速度和最终制动包络的速度，单位mm/s。 *)
    rSaturatedVelocity_mm_s : LREAL;
    (* 上一有效周期速度命令，单位mm/s。 *)
    rPreviousVelocity_mm_s : LREAL;
    (* S_rel制动计算得到的最大向下速度，单位mm/s。 *)
    rStrokeVelocityLimit_mm_s : LREAL;
    (* 当前Profile与机器限值合并后的最大上抬速度绝对值。 *)
    rMaximumUpVelocity_mm_s : LREAL;
    (* 当前Profile、机器和S_rel合并后的最大下压速度绝对值。 *)
    rMaximumDownVelocity_mm_s : LREAL;
    (* 候选Profile与机器限值合并后的最大上抬速度绝对值。 *)
    rCandidateMaximumUpVelocity_mm_s : LREAL;
    (* 候选Profile与机器限值合并后的最大下压速度绝对值。 *)
    rCandidateMaximumDownVelocity_mm_s : LREAL;
    (* 当前Profile与机器限值合并后的最大加速度绝对值。 *)
    rMaximumAcceleration_mm_s2 : LREAL;
    (* Anti-windup积分导数，单位mm/s2。 *)
    rIntegralDerivative_mm_s2 : LREAL;
    (* Z轴绝对软限位跨度，作为S_rel硬上限的配置边界。 *)
    rMaximumRelativeTravel_mm : LREAL;
    (* 机器最大过程力换算值，单位kN。 *)
    rMaximumForce_kN : LREAL;
    (* 最近一次无扰提交的目标S_rel，单位mm。 *)
    rAcceptedTargetRelativePosition_mm : LREAL;
    (* 最近一次无扰提交的硬最大S_rel，单位mm。 *)
    rAcceptedHardMaximumRelativePosition_mm : LREAL;
END_VAR

(* ---------------------------------------------------------
   Z轴导纳力控算法。
   进入：Sequence请求、Force Process Owner和External Active全部成立。
   周期动作：计算Ramp后力误差、PI、Anti-windup、S_rel制动和固定顺序限幅。
   正常出口：发布连续受限速度；不生成P/V/A，不访问轴或MC。
   无效输入：锁存故障并输出零速度，只有显式Reset清除。
   硬边界：禁止继续向下但保留受控上抬能力，并冻结积分。
   --------------------------------------------------------- *)
stOutput.bActive := FALSE;
stOutput.bLimited := FALSE;
stOutput.bAntiWindupFrozen := TRUE;
stOutput.bHardLimitActive := FALSE;
stOutput.bFault := bFaultLatched;
stOutput.nFaultId := udiLatchedFaultId;
stOutput.rVelocityCommand_mm_s := 0.0;
stOutput.rIntegralTerm_mm_s := rIntegralTerm_mm_s;
stOutput.rForceSetRamped_kN := 0.0;
stOutput.rForceError_kN := 0.0;
stOutput.rUnsaturatedVelocity_mm_s := 0.0;
stOutput.rSaturatedVelocity_mm_s := 0.0;
stOutput.rStrokeVelocityLimit_mm_s := 0.0;

IF stInput.bReset THEN
    rIntegralTerm_mm_s := 0.0;
    rPreviousVelocity_mm_s := 0.0;
    rAcceptedTargetRelativePosition_mm := 0.0;
    rAcceptedHardMaximumRelativePosition_mm := 0.0;
    bProfileInitialized := FALSE;
    bFaultLatched := FALSE;
    udiLatchedFaultId := 0;
    stOutput.rIntegralTerm_mm_s := 0.0;
    stOutput.bFault := FALSE;
    stOutput.nFaultId := 0;
    RETURN;
END_IF

IF NOT stInput.bEnable THEN
    rIntegralTerm_mm_s := 0.0;
    rPreviousVelocity_mm_s := 0.0;
    bProfileInitialized := FALSE;
    stOutput.rIntegralTerm_mm_s := 0.0;
    RETURN;
END_IF

IF bFaultLatched THEN
    RETURN;
END_IF

rMaximumRelativeTravel_mm := ABS(stLimits.fZMaxPositionMm - stLimits.fZMinPositionMm);
rMaximumForce_kN := ABS(stLimits.fMaxForceN) * 0.001;
rCandidateMaximumUpVelocity_mm_s := ABS(stProfile.fMaxUpVelocityMmS);
IF ABS(stLimits.fZMaxVelocityMmS) < rCandidateMaximumUpVelocity_mm_s THEN
    rCandidateMaximumUpVelocity_mm_s := ABS(stLimits.fZMaxVelocityMmS);
END_IF
rCandidateMaximumDownVelocity_mm_s := ABS(stProfile.fMaxDownVelocityMmS);
IF ABS(stLimits.fZMaxVelocityMmS) < rCandidateMaximumDownVelocity_mm_s THEN
    rCandidateMaximumDownVelocity_mm_s := ABS(stLimits.fZMaxVelocityMmS);
END_IF

bConfigurationValid := stProfile.bValid
    AND stLimits.bValid
    AND (stProfile.nRevision > 0)
    AND (stInput.rCycleTime_s > 0.0)
    AND (stProfile.fKp >= 0.0)
    AND (stProfile.fKi >= 0.0)
    AND (stProfile.fKaw >= 0.0)
    AND (stProfile.fIntegralLimit >= 0.0)
    AND (stProfile.fMaxUpVelocityMmS > 0.0)
    AND (stProfile.fMaxDownVelocityMmS > 0.0)
    AND (stProfile.fMaxAccelerationMmS2 > 0.0)
    AND (stProfile.fBrakeMarginMm >= 0.0)
    AND (stProfile.fForceRampNS > 0.0)
    AND (stLimits.fZMaxPositionMm > stLimits.fZMinPositionMm)
    AND (stLimits.fZMaxVelocityMmS > 0.0)
    AND (stLimits.fZMaxAccelerationMmS2 > 0.0)
    AND (stLimits.fMaxForceN > 0.0)
    AND (ABS(stProfile.fVelocityFeedForwardMmS) <= ABS(stLimits.fZMaxVelocityMmS))
    AND (stProfile.fIntegralLimit <= ABS(stLimits.fZMaxVelocityMmS))
    AND (stInput.rTargetRelativePosition_mm >= 0.0)
    AND (stInput.rHardMaximumRelativePosition_mm >= stInput.rTargetRelativePosition_mm)
    AND (stInput.rHardMaximumRelativePosition_mm <= rMaximumRelativeTravel_mm)
    AND FC_IsFiniteLReal(rValue := rMaximumRelativeTravel_mm)
    AND FC_IsFiniteLReal(rValue := rMaximumForce_kN)
    AND FC_IsFiniteLReal(rValue := stInput.rCycleTime_s)
    AND FC_IsFiniteLReal(rValue := stProfile.fVelocityFeedForwardMmS)
    AND FC_IsFiniteLReal(rValue := stProfile.fKp)
    AND FC_IsFiniteLReal(rValue := stProfile.fKi)
    AND FC_IsFiniteLReal(rValue := stProfile.fKaw)
    AND FC_IsFiniteLReal(rValue := stProfile.fIntegralLimit)
    AND FC_IsFiniteLReal(rValue := stProfile.fMaxUpVelocityMmS)
    AND FC_IsFiniteLReal(rValue := stProfile.fMaxDownVelocityMmS)
    AND FC_IsFiniteLReal(rValue := stProfile.fMaxAccelerationMmS2)
    AND FC_IsFiniteLReal(rValue := stProfile.fBrakeMarginMm)
    AND FC_IsFiniteLReal(rValue := stProfile.fForceRampNS)
    AND FC_IsFiniteLReal(rValue := stLimits.fZMinPositionMm)
    AND FC_IsFiniteLReal(rValue := stLimits.fZMaxPositionMm)
    AND FC_IsFiniteLReal(rValue := stLimits.fZMaxVelocityMmS)
    AND FC_IsFiniteLReal(rValue := stLimits.fZMaxAccelerationMmS2)
    AND FC_IsFiniteLReal(rValue := stLimits.fMaxForceN);

bInputFinite := FC_IsFiniteLReal(rValue := rForceSetRamped_kN)
    AND FC_IsFiniteLReal(rValue := stInput.rForceSet_kN)
    AND FC_IsFiniteLReal(rValue := stInput.rForceActual_kN)
    AND FC_IsFiniteLReal(rValue := stInput.rRelativePosition_mm)
    AND FC_IsFiniteLReal(rValue := stInput.rTargetRelativePosition_mm)
    AND FC_IsFiniteLReal(rValue := stInput.rHardMaximumRelativePosition_mm)
    AND FC_IsFiniteLReal(rValue := stInput.rTransferVelocity_mm_s)
    AND ((NOT bApplyIntegralPreload)
        OR ((stInput.rTransferVelocity_mm_s >= -rCandidateMaximumUpVelocity_mm_s)
            AND (stInput.rTransferVelocity_mm_s <= rCandidateMaximumDownVelocity_mm_s)))
    AND (rForceSetRamped_kN >= 0.0)
    AND (rForceSetRamped_kN <= ABS(stLimits.fMaxForceN) * 0.001)
    AND (stInput.rForceSet_kN >= 0.0)
    AND (stInput.rForceSet_kN <= ABS(stLimits.fMaxForceN) * 0.001);

IF NOT bConfigurationValid THEN
    bFaultLatched := TRUE;
    udiLatchedFaultId := 16#00008002;
ELSIF NOT bInputFinite THEN
    bFaultLatched := TRUE;
    udiLatchedFaultId := 16#00008003;
ELSIF NOT stInput.bOwnerGranted OR NOT stInput.bExternalActive THEN
    bFaultLatched := TRUE;
    udiLatchedFaultId := 16#00008004;
ELSIF NOT stInput.bForceValid OR NOT stInput.bRelativePositionValid THEN
    bFaultLatched := TRUE;
    udiLatchedFaultId := 16#00008005;
ELSIF bApplyIntegralPreload AND NOT FC_IsFiniteLReal(rValue := rIntegralPreload_mm_s) THEN
    bFaultLatched := TRUE;
    udiLatchedFaultId := 16#00008006;
ELSIF stInput.bBumplessTransfer AND NOT bApplyIntegralPreload THEN
    bFaultLatched := TRUE;
    udiLatchedFaultId := 16#00008007;
END_IF
IF bFaultLatched THEN
    stOutput.bFault := TRUE;
    stOutput.nFaultId := udiLatchedFaultId;
    RETURN;
END_IF

(* 只有有限性和硬范围检查通过后才向ADS诊断发布目标力。 *)
stOutput.rForceSetRamped_kN := rForceSetRamped_kN;

bLimitsMismatch := FALSE;
IF NOT bProfileInitialized THEN
    IF NOT bApplyIntegralPreload THEN
        bFaultLatched := TRUE;
        udiLatchedFaultId := 16#00008009;
    ELSIF stInput.rRelativePosition_mm > stInput.rHardMaximumRelativePosition_mm THEN
        (* 已越过新Profile硬S_rel时禁止作为普通Active恢复。 *)
        bFaultLatched := TRUE;
        udiLatchedFaultId := 16#0000800B;
    ELSE
        stAppliedProfile := stProfile;
        stAppliedLimits := stLimits;
        rAcceptedTargetRelativePosition_mm := stInput.rTargetRelativePosition_mm;
        rAcceptedHardMaximumRelativePosition_mm := stInput.rHardMaximumRelativePosition_mm;
        bProfileInitialized := TRUE;
    END_IF
ELSIF bApplyIntegralPreload THEN
    IF stInput.rRelativePosition_mm > stInput.rHardMaximumRelativePosition_mm THEN
        bFaultLatched := TRUE;
        udiLatchedFaultId := 16#0000800B;
    ELSE
        stAppliedProfile := stProfile;
        stAppliedLimits := stLimits;
        rAcceptedTargetRelativePosition_mm := stInput.rTargetRelativePosition_mm;
        rAcceptedHardMaximumRelativePosition_mm := stInput.rHardMaximumRelativePosition_mm;
    END_IF
ELSE
    bLimitsMismatch := (stLimits.fZMinPositionMm <> stAppliedLimits.fZMinPositionMm)
        OR (stLimits.fZMaxPositionMm <> stAppliedLimits.fZMaxPositionMm)
        OR (stLimits.fZMaxVelocityMmS <> stAppliedLimits.fZMaxVelocityMmS)
        OR (stLimits.fZMaxAccelerationMmS2 <> stAppliedLimits.fZMaxAccelerationMmS2)
        OR (stLimits.fMaxForceN <> stAppliedLimits.fMaxForceN)
        OR (stLimits.bValid <> stAppliedLimits.bValid);
    bProfileMismatch := (stProfile.nRevision <> stAppliedProfile.nRevision)
        OR (stProfile.fVelocityFeedForwardMmS <> stAppliedProfile.fVelocityFeedForwardMmS)
        OR (stProfile.fKp <> stAppliedProfile.fKp)
        OR (stProfile.fKi <> stAppliedProfile.fKi)
        OR (stProfile.fKaw <> stAppliedProfile.fKaw)
        OR (stProfile.fIntegralLimit <> stAppliedProfile.fIntegralLimit)
        OR (stProfile.fMaxUpVelocityMmS <> stAppliedProfile.fMaxUpVelocityMmS)
        OR (stProfile.fMaxDownVelocityMmS <> stAppliedProfile.fMaxDownVelocityMmS)
        OR (stProfile.fMaxAccelerationMmS2 <> stAppliedProfile.fMaxAccelerationMmS2)
        OR (stProfile.fBrakeMarginMm <> stAppliedProfile.fBrakeMarginMm)
        OR (stProfile.fForceRampNS <> stAppliedProfile.fForceRampNS)
        OR (stProfile.bValid <> stAppliedProfile.bValid)
        OR (stInput.rTargetRelativePosition_mm <> rAcceptedTargetRelativePosition_mm)
        OR (stInput.rHardMaximumRelativePosition_mm
            <> rAcceptedHardMaximumRelativePosition_mm)
        OR bLimitsMismatch;
    IF bProfileMismatch THEN
        bFaultLatched := TRUE;
        udiLatchedFaultId := 16#0000800A;
    END_IF
END_IF
IF bFaultLatched THEN
    stOutput.bFault := TRUE;
    stOutput.nFaultId := udiLatchedFaultId;
    RETURN;
END_IF

IF bApplyIntegralPreload THEN
    rIntegralTerm_mm_s := FC_ClampLReal(
        rValue := rIntegralPreload_mm_s,
        rMinimum := -ABS(stAppliedProfile.fIntegralLimit),
        rMaximum := ABS(stAppliedProfile.fIntegralLimit));
    rPreviousVelocity_mm_s := stInput.rTransferVelocity_mm_s;
END_IF

rForceError_kN := rForceSetRamped_kN - stInput.rForceActual_kN;
rUnsaturatedVelocity_mm_s := stAppliedProfile.fVelocityFeedForwardMmS
    + stAppliedProfile.fKp * rForceError_kN
    + rIntegralTerm_mm_s;
IF NOT FC_IsFiniteLReal(rValue := rUnsaturatedVelocity_mm_s) THEN
    bFaultLatched := TRUE;
    udiLatchedFaultId := 16#00008008;
    stOutput.bFault := TRUE;
    stOutput.nFaultId := udiLatchedFaultId;
    RETURN;
END_IF

(* LIMIT_STAGE_PROFILE：先执行Profile上下速度限幅。 *)
rBoundaryLimitedVelocity_mm_s := FC_ClampLReal(
    rValue := rUnsaturatedVelocity_mm_s,
    rMinimum := -ABS(stAppliedProfile.fMaxUpVelocityMmS),
    rMaximum := ABS(stAppliedProfile.fMaxDownVelocityMmS));

(* LIMIT_STAGE_MACHINE：再执行机器最大速度限幅。 *)
rMaximumUpVelocity_mm_s := ABS(stAppliedProfile.fMaxUpVelocityMmS);
IF ABS(stLimits.fZMaxVelocityMmS) < rMaximumUpVelocity_mm_s THEN
    rMaximumUpVelocity_mm_s := ABS(stLimits.fZMaxVelocityMmS);
END_IF
rMaximumDownVelocity_mm_s := ABS(stAppliedProfile.fMaxDownVelocityMmS);
IF ABS(stLimits.fZMaxVelocityMmS) < rMaximumDownVelocity_mm_s THEN
    rMaximumDownVelocity_mm_s := ABS(stLimits.fZMaxVelocityMmS);
END_IF
rBoundaryLimitedVelocity_mm_s := FC_ClampLReal(
    rValue := rBoundaryLimitedVelocity_mm_s,
    rMinimum := -rMaximumUpVelocity_mm_s,
    rMaximum := rMaximumDownVelocity_mm_s);

rMaximumAcceleration_mm_s2 := ABS(stAppliedProfile.fMaxAccelerationMmS2);
IF ABS(stLimits.fZMaxAccelerationMmS2) < rMaximumAcceleration_mm_s2 THEN
    rMaximumAcceleration_mm_s2 := ABS(stLimits.fZMaxAccelerationMmS2);
END_IF
(* EFFECTIVE_DECELERATION_READY：制动包络和Rate Limit必须使用同一有效加减速度。 *)

(* LIMIT_STAGE_SREL_BRAKE：按S_rel剩余行程计算向下制动限速。 *)
rStrokeVelocityLimit_mm_s := FC_CalcStrokeVelocityLimit(
    rRemainingStroke_mm := stInput.rTargetRelativePosition_mm
        - stInput.rRelativePosition_mm,
    rBrakeMargin_mm := stAppliedProfile.fBrakeMarginMm,
    rMaximumDeceleration_mm_s2 := rMaximumAcceleration_mm_s2);
IF NOT FC_IsFiniteLReal(rValue := rStrokeVelocityLimit_mm_s) THEN
    bFaultLatched := TRUE;
    udiLatchedFaultId := 16#0000800D;
    stOutput.bFault := TRUE;
    stOutput.nFaultId := udiLatchedFaultId;
    RETURN;
END_IF
IF rStrokeVelocityLimit_mm_s < rMaximumDownVelocity_mm_s THEN
    rMaximumDownVelocity_mm_s := rStrokeVelocityLimit_mm_s;
END_IF
IF rBoundaryLimitedVelocity_mm_s > rMaximumDownVelocity_mm_s THEN
    rBoundaryLimitedVelocity_mm_s := rMaximumDownVelocity_mm_s;
END_IF

bHardLimitActive := stInput.bHardForceActive
    OR (ABS(stInput.rForceActual_kN * 1000.0) >= ABS(stLimits.fMaxForceN))
    OR stInput.bHardStrokeActive
    OR (stInput.rRelativePosition_mm >= stInput.rHardMaximumRelativePosition_mm)
    OR stInput.bCollisionLimitActive;
bDownwardBoundaryActive := stInput.bHardStrokeActive
    OR (stInput.rRelativePosition_mm >= stInput.rHardMaximumRelativePosition_mm);

(* LIMIT_STAGE_HARD_BOUNDARY：Secondary/Hard边界禁止继续向下。 *)
IF stInput.bHardForceActive
    OR (ABS(stInput.rForceActual_kN * 1000.0) >= ABS(stLimits.fMaxForceN))
    OR bDownwardBoundaryActive THEN
    IF rBoundaryLimitedVelocity_mm_s > 0.0 THEN
        rBoundaryLimitedVelocity_mm_s := 0.0;
    END_IF
    rMaximumDownVelocity_mm_s := 0.0;
END_IF

(* LIMIT_STAGE_COLLISION：Collision边界同样只封锁向下方向。 *)
IF stInput.bCollisionLimitActive THEN
    IF rBoundaryLimitedVelocity_mm_s > 0.0 THEN
        rBoundaryLimitedVelocity_mm_s := 0.0;
    END_IF
    rMaximumDownVelocity_mm_s := 0.0;
END_IF

IF bHardLimitActive AND (rPreviousVelocity_mm_s > 0.0) THEN
    (* 已到硬边界时不得由后续加速度限幅继续保留向下速度。 *)
    rPreviousVelocity_mm_s := 0.0;
END_IF

(* LIMIT_STAGE_ACCELERATION：最后执行速度变化率/最大加速度限幅。 *)
rSaturatedVelocity_mm_s := FC_LimitRate(
    rCurrent := rPreviousVelocity_mm_s,
    rTarget := rBoundaryLimitedVelocity_mm_s,
    rRateUpPer_s := rMaximumAcceleration_mm_s2,
    rRateDownPer_s := rMaximumAcceleration_mm_s2,
    rCycleTime_s := stInput.rCycleTime_s);
IF NOT FC_IsFiniteLReal(rValue := rSaturatedVelocity_mm_s) THEN
    bFaultLatched := TRUE;
    udiLatchedFaultId := 16#0000800E;
    stOutput.bFault := TRUE;
    stOutput.nFaultId := udiLatchedFaultId;
    RETURN;
END_IF

bEnvelopeViolation := (rSaturatedVelocity_mm_s > rMaximumDownVelocity_mm_s)
    OR (rSaturatedVelocity_mm_s < -rMaximumUpVelocity_mm_s);
IF rSaturatedVelocity_mm_s > rMaximumDownVelocity_mm_s THEN
    (* Rate Limit不得重新越过当前S_rel制动包络。 *)
    rSaturatedVelocity_mm_s := rMaximumDownVelocity_mm_s;
ELSIF rSaturatedVelocity_mm_s < -rMaximumUpVelocity_mm_s THEN
    (* 无扰预置和Rate Limit同样不得越过上抬速度硬包络。 *)
    rSaturatedVelocity_mm_s := -rMaximumUpVelocity_mm_s;
END_IF

bErrorRequestsDownward := rForceError_kN > 0.0;
bFreezeIntegral := bHardLimitActive
    OR bEnvelopeViolation
    OR (bErrorRequestsDownward AND (rMaximumDownVelocity_mm_s <= 0.0));

IF bApplyIntegralPreload THEN
    bFreezeIntegral := TRUE;
ELSIF NOT bFreezeIntegral THEN
    rIntegralDerivative_mm_s2 := stAppliedProfile.fKi * rForceError_kN
        + stAppliedProfile.fKaw * (rSaturatedVelocity_mm_s - rUnsaturatedVelocity_mm_s);
    IF NOT FC_IsFiniteLReal(rValue := rIntegralDerivative_mm_s2) THEN
        bFaultLatched := TRUE;
        udiLatchedFaultId := 16#0000800F;
        stOutput.bFault := TRUE;
        stOutput.nFaultId := udiLatchedFaultId;
        RETURN;
    END_IF
    rUpdatedIntegralTerm_mm_s := rIntegralTerm_mm_s
        + rIntegralDerivative_mm_s2 * stInput.rCycleTime_s;
    IF NOT FC_IsFiniteLReal(rValue := rUpdatedIntegralTerm_mm_s) THEN
        bFaultLatched := TRUE;
        udiLatchedFaultId := 16#00008010;
        stOutput.bFault := TRUE;
        stOutput.nFaultId := udiLatchedFaultId;
        RETURN;
    END_IF
    rIntegralTerm_mm_s := FC_ClampLReal(
        rValue := rUpdatedIntegralTerm_mm_s,
        rMinimum := -ABS(stAppliedProfile.fIntegralLimit),
        rMaximum := ABS(stAppliedProfile.fIntegralLimit));
    IF NOT FC_IsFiniteLReal(rValue := rIntegralTerm_mm_s) THEN
        bFaultLatched := TRUE;
        udiLatchedFaultId := 16#00008011;
        stOutput.bFault := TRUE;
        stOutput.nFaultId := udiLatchedFaultId;
        RETURN;
    END_IF
END_IF

IF bEnvelopeViolation THEN
    (* 包络突变意味着目标或测量无法按配置减速度无扰跟随。 *)
    bFaultLatched := TRUE;
    udiLatchedFaultId := 16#0000800C;
    (* 故障扫描不得发布可被后续轨迹层消费的非零速度。 *)
    rSaturatedVelocity_mm_s := 0.0;
    stOutput.bActive := FALSE;
END_IF

stOutput.rVelocityCommand_mm_s := rSaturatedVelocity_mm_s;
stOutput.rIntegralTerm_mm_s := rIntegralTerm_mm_s;
stOutput.rForceSetRamped_kN := rForceSetRamped_kN;
stOutput.rForceError_kN := rForceError_kN;
stOutput.rUnsaturatedVelocity_mm_s := rUnsaturatedVelocity_mm_s;
stOutput.rSaturatedVelocity_mm_s := rSaturatedVelocity_mm_s;
stOutput.rStrokeVelocityLimit_mm_s := rStrokeVelocityLimit_mm_s;
stOutput.bActive := NOT bFaultLatched;
stOutput.bLimited := ABS(rSaturatedVelocity_mm_s - rUnsaturatedVelocity_mm_s) > 0.000000001;
stOutput.bAntiWindupFrozen := bFreezeIntegral;
stOutput.bHardLimitActive := bHardLimitActive;
stOutput.bFault := bFaultLatched;
stOutput.nFaultId := udiLatchedFaultId;
rPreviousVelocity_mm_s := rSaturatedVelocity_mm_s;

END_FUNCTION_BLOCK

// ---- POUs/Functions/FC_CalcStrokeVelocityLimit.TcPOU
FUNCTION FC_CalcStrokeVelocityLimit : LREAL
VAR_INPUT
    (* 距离几何边界的剩余正向行程，单位毫米。 *)
    rRemainingStroke_mm : LREAL;
    (* 在边界前保留的制动裕量，单位毫米。 *)
    rBrakeMargin_mm : LREAL;
    (* 允许的最大减速度，单位毫米每二次方秒。 *)
    rMaximumDeceleration_mm_s2 : LREAL;
END_VAR
VAR
    (* 扣除制动裕量后的可用行程，单位毫米。 *)
    rUsableStroke_mm : LREAL;
END_VAR

IF (rRemainingStroke_mm <= rBrakeMargin_mm)
    OR (rBrakeMargin_mm < 0.0)
    OR (rMaximumDeceleration_mm_s2 <= 0.0)
    OR NOT FC_IsFiniteLReal(rValue := rRemainingStroke_mm)
    OR NOT FC_IsFiniteLReal(rValue := rBrakeMargin_mm)
    OR NOT FC_IsFiniteLReal(rValue := rMaximumDeceleration_mm_s2) THEN
    (* 已到边界或减速度无效时，向边界方向速度上限必须为零。 *)
    FC_CalcStrokeVelocityLimit := 0.0;
    RETURN;
END_IF

rUsableStroke_mm := rRemainingStroke_mm - rBrakeMargin_mm;
FC_CalcStrokeVelocityLimit := SQRT(2.0 * rMaximumDeceleration_mm_s2 * rUsableStroke_mm);

END_FUNCTION

// ---- POUs/FunctionBlocks/Control/FB_ZExternalTrajectory.TcPOU
FUNCTION_BLOCK FB_ZExternalTrajectory
VAR_INPUT
    (* 调用者完整赋值的External轨迹输入快照。 *)
    stInput : ST_ZExternalTrajectoryInput;
END_VAR
VAR_OUTPUT
    (* 仅由已接受设定值推导的轨迹包和状态。 *)
    stOutput : ST_ZExternalTrajectoryOutput;
END_VAR
VAR
    (* 当前纯轨迹状态。 *)
    eState : E_ZExternalTrajectoryState;
    (* 最近一次已处理的Adapter接受周期计数。 *)
    udiLastAcceptedFeedCycleCounter : UDINT;
    (* 最近一次发布的位置，单位mm。 *)
    rLastPublishedPosition_mm : LREAL;
    (* 最近一次发布的速度，单位mm/s。 *)
    rLastPublishedVelocity_mm_s : LREAL;
    (* 最近一次发布的加速度，单位mm/s2。 *)
    rLastPublishedAcceleration_mm_s2 : LREAL;
    (* 最近一次发布的方向。 *)
    nLastPublishedDirection : DINT;
    (* 最近一次发布包携带的Hard Inhibit连续性绕过标志。 *)
    bLastPublishedPositiveMotionInhibited : BOOL;
    (* 最近一次有效的非零方向。 *)
    nLastNonZeroDirection : DINT;
    (* 零速换向完成后待预置的新方向。 *)
    nPendingDirection : DINT;
    (* 当前静止握手状态已经确认的接受周期数。 *)
    nAcceptedStateCycles : UINT;
    (* 当前External Active生命周期已经同步接受基准。 *)
    bInitialized : BOOL;
    (* 本扫描收到一个新的Adapter接受确认。 *)
    bNewAcceptedFeed : BOOL;
    (* 本扫描接受的是最近一次发布的零速包。 *)
    bAcceptedPublishedZero : BOOL;
    (* 配置、周期和目标满足纯算法边界。 *)
    bConfigurationValid : BOOL;
    (* 已接受P/V/A均有限且位于速度和加速度边界内。 *)
    bAcceptedMotionValid : BOOL;
    (* 新接受包与最近一次发布包连续。 *)
    bAcceptedContinuityValid : BOOL;
    (* 当前目标速度对应的离散方向。 *)
    nTargetDirection : DINT;
    (* 本扫描Rate Limit结果，单位mm/s。 *)
    rNextVelocity_mm_s : LREAL;
    (* 本扫描梯形积分加速度，单位mm/s2。 *)
    rNextAcceleration_mm_s2 : LREAL;
    (* 本扫描梯形积分位置，单位mm。 *)
    rNextPosition_mm : LREAL;
    (* 算法故障锁存。 *)
    bFaultLatched : BOOL;
    (* 首次锁存的确定性故障编号。 *)
    udiLatchedFaultId : UDINT;
END_VAR

